(* IEC 61131-3 sources: elnaProjects/ElpcLogic/PomarKc7Changed/build_USO_ecl/_ (part 5) *)

FUNCTION_BLOCK fb_vibegPNSAlg
  VAR_IN_OUT
    StrAlg : struct_Alg;
  END_VAR
  VAR
    autoPnsOff : struct_PhaseAlgoritm;
    waitVibeg : struct_PhaseAlgoritm;
    pnsOff : struct_PhaseAlgoritm;
    vibegEnd : struct_PhaseAlgoritm;
  END_VAR
  VAR_IN_OUT
    algContinue : struct_Question;
  END_VAR
  VAR
    fb_autoPnsOff : fb_ph_algoritm;
    fb_waitVibeg : fb_ph_Timer;
    fb_algContinue : fb_Question;
    fb_pnsOff : fb_ph_Switch;
    fb_vibegEnd : fb_ph_CustomPhase;
    _sunpackerCommand : fb_sunpackerCommand;
    _statusAi : TYPE_StatusAi;
    _Answers : TYPE_Answers;
    _statusDualInput : TYPE_statusDualInput;
    _DualStateImAction : TYPE_DualStateImAction;
    _PhaseAlgoritmAction : TYPE_PhaseAlgoritmAction;
    source : BYTE;
    cmd : BYTE;
    lastCmd : BYTE;
    source_for_Status : BYTE;
    cmd_for_Status : BYTE;
    command_error_for_Status : BYTE;
    resetCmdTimer : TON;
    resetCmdTimerPriznak : BOOL;
    onInit : BOOL;
    waitReset : TON;
  END_VAR
  VAR_EXTERNAL
    IM : ImConfig;
    algoritms : AlgoritmsConfig;
    ai : AiConfig;
    protections : ProtectionsConfig;
    AlgTimers : struct_AlgTimers;
  END_VAR

  IF NOT onInit THEN
   fb_autoPnsOff(phaseNumber:=0, act:=_reset, waitCompletion:=FALSE);
    fb_waitVibeg(phaseNumber:=1, delay:=T#300S);
       algContinue.AnswerVariants:=_Answers.ANS_YES;
       fb_pnsOff(phaseNumber:=2, act:=_off);
     fb_vibegEnd(phaseNumber:=14);
  onInit:=TRUE;
  END_IF;

   fb_autoPnsOff(StrPh:=autoPnsOff, alg:=algoritms.autoPns);
    fb_waitVibeg(StrPh:=waitVibeg, timer:=AlgTimers.vibegPNS_Timer);
  fb_algContinue(StrQ:=algContinue);
       fb_pnsOff(StrPh:=pnsOff, Im:=IM.pns);
     fb_vibegEnd(StrPh:=vibegEnd);

  IF StrAlg.isRuning THEN

  StrAlg.hasError := autoPnsOff.error OR pnsOff.error;

      IF IM.pns.onStatus = _statusDualInput.STATUS_ON AND NOT vibegEnd.top THEN

  	runPhase(vibegEnd);
            runPhase(waitVibeg);
            askQuestion(algContinue);

      END_IF;

      IF waitVibeg.top OR (algContinue.answer = _Answers.ANS_YES) THEN
  	vibegEnd.top:=TRUE;
  	resetPhase(waitVibeg);
            resetQuestion(algContinue);

            resetAiProtection(protections.Os_sdvig_nagnetatelja_minus);
            (*resetDiProtection(protections.Vibro_skorost_OP_shesterni_RED_T6);*)

  	(*IM.SingleSignals.P_oil_low.Disabled_Sig:=TRUE;*)
  	ai.Pmasla_posle_GNS.Disabled_LA:=TRUE;
            ai.Pmasla_posle_GNS.Disabled_LW:=TRUE;
            ai.Pmasla_posle_NU.Disabled_LW:=TRUE;
  	runPhase(pnsOff);
      END_IF;

      StrAlg.isEnded:=pnsOff.top;

  END_IF;

  StrAlg.CanRun := StrAlg.inCanRun;
  StrAlg.OpcCommandsDisabled := StrAlg.inOpcCommandsDisabled;

  (* ---- Если управление с ВУ заблокировано, то  передаем команду из алгоритма ---- *)
  IF StrAlg.inOpcCommandsDisabled THEN
  	StrAlg.inCommand := StrAlg.inCommand_Alg;
  ELSE (* иначе передаем команду с АРМа*)
  	StrAlg.inCommand := StrAlg.inCommand_ARM;
  END_IF;

  _sunpackerCommand(command := StrAlg.inCommand);
  	source := _sunpackerCommand.source;
  	cmd := _sunpackerCommand.cmd;

  IF cmd <> 0 AND lastCmd <> cmd AND (((NOT StrAlg.opcCommandsDisabled) AND source > 0) OR source = 0) then
  	CASE BYTE_TO_INT(cmd) OF
  		(*cmdRun*) 1: 	IF (StrAlg.CanRun) THEN
  					StrAlg.isRuning := TRUE;
  					StrAlg.isEnded := FALSE;
  					StrAlg.hasError := FALSE;
  					(*****************       OnRun       *****************)
                                                    runPhase(autoPnsOff);

  					cmd_for_Status := cmd;
  					source_for_Status := source;
  					command_error_for_Status := 0;
  				ELSE
  					StrAlg.isRuning := FALSE;
  					StrAlg.isEnded := FALSE;
  					StrAlg.hasError 	:= FALSE;

  					cmd_for_Status := 0;
  					source_for_Status := source;
  					command_error_for_Status := cmd;
  				END_IF;
  		(*cmdReset*) 2: 	StrAlg.isRuning := FALSE;
  				StrAlg.isEnded := FALSE;
  				StrAlg.hasError 	:= FALSE;

                                           (*****************       OnReset       *****************)
                                         waitReset(IN:=FALSE);
                                         resetPhase(autoPnsOff);
                                         resetPhase(waitVibeg);
                                         resetPhase(vibegEnd);
                                         resetPhase(pnsOff);
                                         resetQuestion(algContinue);

  				cmd_for_Status := cmd;
  				source_for_Status := source;
  				command_error_for_Status := 0;
  	END_CASE;
  	resetCmdTimer(IN := false);
  	resetCmdTimerPriznak := TRUE;
  END_IF;
  lastCmd := cmd;

  resetCmdTimer(IN := resetCmdTimerPriznak, PT := T#5S);
  IF resetCmdTimer.Q THEN
  	resetCmdTimerPriznak := FALSE;
  	source_for_Status := 0;
  	cmd_for_Status := 0;
  	command_error_for_Status := 0;
  END_IF;

  StrAlg.Start:= autoPnsOff.startStatus
              OR waitVibeg.startStatus
              OR pnsOff.startStatus
              OR vibegEnd.startStatus;

  StrAlg.Error:= autoPnsOff.errorStatus
              OR waitVibeg.errorStatus
              OR pnsOff.errorStatus
              OR vibegEnd.errorStatus;

  StrAlg.Top:=   autoPnsOff.topStatus
              OR waitVibeg.topStatus
              OR pnsOff.topStatus
              OR vibegEnd.topStatus;

  (*TODO: TYPE PROGRAM CODE HERE*)
  StrAlg.status :=  SHL(BYTE_TO_DWORD(source_for_Status), 29)
  			OR SHL(BYTE_TO_DWORD(cmd_for_Status), 26)
  			OR SHL(BYTE_TO_DWORD(command_error_for_Status), 23)
  			OR SHL(BOOL_TO_DWORD(StrAlg.OpcCommandsDisabled ), 21)
  			OR SHL(BOOL_TO_DWORD(StrAlg.hasError),4)
  			OR SHL(BOOL_TO_DWORD(StrAlg.CanRun),2)
  			OR SHL(BOOL_TO_DWORD(StrAlg.isEnded),1)
  			OR BOOL_TO_DWORD(StrAlg.isRuning);
END_FUNCTION_BLOCK

FUNCTION_BLOCK fb_AutoNUAlg
  VAR_IN_OUT
    StrAlg : struct_Alg;
    nu1 : struct_OilPump;
    nu2 : struct_OilPump;
  END_VAR
  VAR_INPUT
    dPoil : struct_AI;
  END_VAR
  VAR_IN_OUT
    mainNU : struct_DiscretParametr;
    Lowdp_di : struct_singleSignal;
    Ust_Swap : struct_AnalogParametr;
  END_VAR
  VAR
    _prevMainNU : UINT;
    _sunpackerCommand : fb_sunpackerCommand;
    _statusAi : TYPE_StatusAi;
    _statusDualInput : TYPE_statusDualInput;
    _commandDualInput : TYPE_commandDualInput;
    source : BYTE;
    cmd : BYTE;
    lastCmd : BYTE;
    source_for_Status : BYTE;
    cmd_for_Status : BYTE;
    command_error_for_Status : BYTE;
    resetCmdTimer : TON;
    waitPressure : TON;
    waitPressureTrig : R_TRIG;
    resetCmdTimerPriznak : BOOL;
    onInit : BOOL;
    onStart : BOOL;
  END_VAR
  VAR_EXTERNAL
    NotHasRezervNU : BOOL;
    Reset_HasNU : BOOL;
  END_VAR

  IF NOT onInit THEN
  StrAlg.inCanRun:=TRUE;
  StrAlg.inOpcCommandsDisabled:=TRUE;
  (*nu1.Osnovnoy:=TRUE; nu2.Osnovnoy:=FALSE;*)
  onInit:=TRUE;
  END_IF;

  IF Reset_HasNU THEN
  nu1.inBlocked:=FALSE;
  nu2.inBlocked:=FALSE;
  END_IF;

  NotHasRezervNU:=(nu1.Blocked OR nu2.Blocked);

  IF StrAlg.isRuning THEN

  StrAlg.hasError := nu1.CommandFault OR nu2.CommandFault OR (dPoil.interval<_statusAi.normal);

   IF mainNU.value<>_prevMainNU OR NOT onStart THEN

          CASE mainNU.value OF
  	0: nu1.Osnovnoy:=TRUE; nu2.Osnovnoy:=FALSE;
  	1: nu1.Osnovnoy:=FALSE; nu2.Osnovnoy:=TRUE;

          END_CASE;

      IF  nu1.Osnovnoy AND NOT nu1.Blocked THEN
          nu1.inCommand_Alg:=BYTE_TO_WORD(_commandDualInput.CMD_ON);
      ELSIF NOT NotHasRezervNU THEN
          nu1.inCommand_Alg:=BYTE_TO_WORD(_commandDualInput.CMD_OFF);
      END_IF;

      IF  nu2.Osnovnoy AND NOT nu2.Blocked THEN
          nu2.inCommand_Alg:=BYTE_TO_WORD(_commandDualInput.CMD_ON);
       ELSIF NOT NotHasRezervNU THEN
          nu2.inCommand_Alg:=BYTE_TO_WORD(_commandDualInput.CMD_OFF);
      END_IF;
        onStart:=TRUE;
       _prevMainNU:=mainNU.value;
   END_IF;

    (*IF (nu1.onStatus = _statusDualInput.STATUS_On) OR (nu2.onStatus = _statusDualInput.STATUS_On) THEN*)
      (*Если через 5С насос не нагнал 100кПа масла - он сломался и надо переключить насос*)
      IF dPoil.interval>= _statusAi.NORMAL THEN
            waitPressure(IN:=(dPoil.value<Ust_Swap.Value OR LowdP_DI.q) AND NOT NotHasRezervNU, PT:= T#5S);
      ELSE
  	waitPressure(IN:=(FALSE));
      END_IF;

      waitPressureTrig(CLK:=waitPressure.Q);
      IF waitPressureTrig.Q THEN
  	(*IF nu1.onStatus = _statusDualInput.STATUS_ON THEN*)
             IF mainNU.value = 0 THEN
  		nu1.inBlocked:=TRUE;
                      nu1.inCommand_Alg:=BYTE_TO_WORD(_commandDualInput.CMD_OFF);
  			(*IF 	mainNU.value = 0 THEN*)
                                          setValue(mainNU, 1);
  			(*END_IF;*)
  	END_IF;

  	(*IF nu2.onStatus = _statusDualInput.STATUS_ON THEN*)
            IF mainNU.value = 1 THEN
  		nu2.inBlocked:=TRUE;
                      nu2.inCommand_Alg:=BYTE_TO_WORD(_commandDualInput.CMD_OFF);
  			(*IF 	mainNU.value = 1 THEN*)
  				setValue(mainNU, 0);
  			(*END_IF;*)
  	END_IF;
      END_IF;
   (* END_IF;*)

  END_IF;

  StrAlg.CanRun := StrAlg.inCanRun;

  StrAlg.OpcCommandsDisabled := StrAlg.inOpcCommandsDisabled;

  (* ---- Если управление с ВУ заблокировано, то  передаем команду из алгоритма ---- *)
  IF StrAlg.inOpcCommandsDisabled THEN
  	StrAlg.inCommand := StrAlg.inCommand_Alg;
  ELSE (* иначе передаем команду с АРМа*)
  	StrAlg.inCommand := StrAlg.inCommand_ARM;
  END_IF;

  _sunpackerCommand(command := StrAlg.inCommand);
  	source := _sunpackerCommand.source;
  	cmd := _sunpackerCommand.cmd;

  IF cmd <> 0 AND lastCmd <> cmd AND (((NOT StrAlg.opcCommandsDisabled) AND source > 0) OR source = 0) then
  	CASE BYTE_TO_INT(cmd) OF
  		(*cmdRun*) 1: 	IF (StrAlg.CanRun) THEN
  					StrAlg.isRuning := TRUE;
  					StrAlg.isEnded := FALSE;
  					StrAlg.hasError := FALSE;

                                                    (*****************       OnRun       *****************)
  					nu1.inOpcCommandsDisabled:=TRUE;
                                                    nu2.inOpcCommandsDisabled:=TRUE;

  					cmd_for_Status := cmd;
  					source_for_Status := source;
  					command_error_for_Status := 0;
  				ELSE
  					StrAlg.isRuning := FALSE;
  					StrAlg.isEnded := FALSE;
  					StrAlg.hasError 	:= FALSE;

  					cmd_for_Status := 0;
  					source_for_Status := source;
  					command_error_for_Status := cmd;
  				END_IF;
  		(*cmdReset*) 2: 	StrAlg.isRuning := FALSE;
  				StrAlg.isEnded := FALSE;
  				StrAlg.hasError 	:= FALSE;

                                          (*****************       OnReset       *****************)
                                          waitPressure(IN:=(FALSE));
                                          onStart:=FALSE;

  				cmd_for_Status := cmd;
  				source_for_Status := source;
  				command_error_for_Status := 0;
  	END_CASE;
  	resetCmdTimer(IN := false);
  	resetCmdTimerPriznak := TRUE;
  END_IF;
  lastCmd := cmd;

  resetCmdTimer(IN := resetCmdTimerPriznak, PT := T#5S);
  IF resetCmdTimer.Q THEN
  	resetCmdTimerPriznak := FALSE;
  	source_for_Status := 0;
  	cmd_for_Status := 0;
  	command_error_for_Status := 0;
  END_IF;

  (*TODO: TYPE PROGRAM CODE HERE*)
  StrAlg.status :=  SHL(BYTE_TO_DWORD(source_for_Status), 29)
  			OR SHL(BYTE_TO_DWORD(cmd_for_Status), 26)
  			OR SHL(BYTE_TO_DWORD(command_error_for_Status), 23)
  			OR SHL(BOOL_TO_DWORD(StrAlg.OpcCommandsDisabled ), 21)
                                OR SHL(BOOL_TO_DWORD(NotHasRezervNU), 15)
  			OR SHL(BOOL_TO_DWORD(StrAlg.hasError),4)
  			OR SHL(BOOL_TO_DWORD(StrAlg.CanRun),2)
  			OR SHL(BOOL_TO_DWORD(StrAlg.isEnded),1)
  			OR BOOL_TO_DWORD(StrAlg.isRuning);
END_FUNCTION_BLOCK

FUNCTION_BLOCK fb_ph_WaitAnalogValue
  VAR_IN_OUT
    ai : struct_AI;
  END_VAR
  VAR_INPUT
    more : LREAL;
    less : LREAL;
    PhaseNumber : UINT;
  END_VAR
  VAR_IN_OUT
    StrPh : struct_PhaseAlgoritm;
  END_VAR
  VAR
    CommandFault_Trig : R_TRIG;
    reset_Trig : R_TRIG;
    _statusAi : TYPE_StatusAi;
    _statusDualInput : TYPE_statusDualInput;
  END_VAR

  IF StrPh.run AND NOT StrPh.start THEN
  	StrPh.start := TRUE;
  	StrPh.top := FALSE;
  	StrPh.error := FALSE;
            StrPh.run:=FALSE;
  END_IF;

  IF StrPh.start AND NOT StrPh.top THEN
                      IF ai.interval < _statusAi.normal THEN
  	              StrPh.error := TRUE;
                          StrPh.top:=FALSE;
                      ELSE
                              IF (more<>0.0) OR (less<>0.0) THEN
                              StrPh.top:=TRUE;
  	                    IF more<>0.0 THEN StrPh.top:=StrPh.top AND (ai.value > more); END_IF;
  	                    IF less<>0.0 THEN StrPh.top:=StrPh.top AND (ai.value < less); END_IF;
                              ELSE
  	                  StrPh.top:=TRUE;
                              END_IF;
                     END_IF;
  END_IF;

  IF StrPh.top THEN
  StrPh.error := FALSE;
  END_IF;

  reset_Trig(CLK := StrPh.reset);
  IF reset_Trig.Q THEN
  	StrPh.start := FALSE;
  	StrPh.error := FALSE;
  	StrPh.top := FALSE;
            StrPh.run:=FALSE;
            StrPh.reset:=FALSE;
  END_IF;

  StrPh.startStatus := SHL(BOOL_TO_DWORD(StrPh.start), PhaseNumber);
  StrPh.errorStatus := SHL(BOOL_TO_DWORD(StrPh.error), PhaseNumber);
  StrPh.topStatus := SHL(BOOL_TO_DWORD(StrPh.top), PhaseNumber);
END_FUNCTION_BLOCK

FUNCTION resetAndDisable : BOOL
  VAR_IN_OUT
    alg : struct_Alg;
  END_VAR
  VAR CONSTANT
    cmdReset : WORD      := 2;
  END_VAR

  IF alg.isRuning THEN
                      alg.inOpcCommandsDisabled:=TRUE;
  		alg.inCommand_Alg:=cmdReset;
  END_IF;

   alg.inCanRun:=FALSE;
END_FUNCTION

FUNCTION_BLOCK fb_puskOilSystemAlg
  VAR_IN_OUT
    StrAlg : struct_Alg;
  END_VAR
  VAR
    pnsOn : struct_PhaseAlgoritm;
    LowOil : struct_PhaseAlgoritm;
    BreakPuskTimer_Poil : struct_PhaseAlgoritm;
    Poil_DefenseActive : struct_PhaseAlgoritm;
    autoNuOn : struct_PhaseAlgoritm;
    nuOn : struct_PhaseAlgoritm;
    nu1On : struct_PhaseAlgoritm;
    nu2On : struct_PhaseAlgoritm;
    di_dPmg : struct_PhaseAlgoritm;
    dP_oilGas100 : struct_PhaseAlgoritm;
    runProtect_dP : struct_PhaseAlgoritm;
    testUnsuccessful : struct_PhaseAlgoritm;
    fb_pnsOn : fb_ph_Switch;
    fb_LowOil : fb_ph_WaitAnalogValue;
    fb_BreakPuskTimer_Poil : fb_ph_Timer;
    fb_Poil_DefenseActive : fb_ph_CustomPhase;
    fb_nuOn : fb_ph_CustomPhase;
    fb_nu1On : fb_ph_OilPump;
    fb_nu2On : fb_ph_OilPump;
    fb_autoNuOn : fb_ph_algoritm;
    fb_di_dPmg : fb_ph_CustomPhase;
    fb_dP_oilGas100 : fb_ph_WaitAnalogValue;
    fb_runProtect_dP : fb_ph_CustomPhase;
    fb_testUnsuccessful : fb_ph_CustomPhase;
    _sunpackerCommand : fb_sunpackerCommand;
    _statusAi : TYPE_StatusAi;
    _Answers : TYPE_Answers;
    _statusDualInput : TYPE_statusDualInput;
    _DualStateImAction : TYPE_DualStateImAction;
    _PhaseAlgoritmAction : TYPE_PhaseAlgoritmAction;
    source : BYTE;
    cmd : BYTE;
    lastCmd : BYTE;
    source_for_Status : BYTE;
    cmd_for_Status : BYTE;
    command_error_for_Status : BYTE;
    resetCmdTimer : TON;
    resetCmdTimerPriznak : BOOL;
    onInit : BOOL;
    waitReset : TON;
  END_VAR
  VAR_EXTERNAL
    IM : ImConfig;
    algoritms : AlgoritmsConfig;
    ai : AiConfig;
    protections : ProtectionsConfig;
    AlgTimers : struct_AlgTimers;
  END_VAR

  IF NOT onInit THEN
                 fb_pnsOn(phaseNumber:=0, act:=_on);
                fb_LowOil(phaseNumber:=1);
   fb_BreakPuskTimer_Poil(phaseNumber:=3, delay:=T#240S);
    fb_Poil_DefenseActive(phaseNumber:=5);
                  fb_nuOn(phaseNumber:=6);
                 fb_nu1On(phaseNumber:=11, act:=_on);
                 fb_nu2On(phaseNumber:=12, act:=_on);
              fb_autoNuOn(phaseNumber:=7, act:=_run, waitCompletion:=FALSE);
               fb_di_dPmg(phaseNumber:=8);
          fb_dP_oilGas100(phaseNumber:=9);
         fb_runProtect_dP(phaseNumber:=10);
      fb_testUnsuccessful(phaseNumber:=17);

  onInit:=TRUE;
  END_IF;

                fb_pnsOn(StrPh:=pnsOn, Im:=IM.pns);
               (*fb_LowOil(StrPh:=LowOil, ai:=ai.Pmasla_posle_GNS, more:=im.AutoPns_UstRun.Value);*)
  fb_BreakPuskTimer_Poil(StrPh:=BreakPuskTimer_Poil, timer:=AlgTimers.puskOilSystem_BreakPuskTimer_Poil);
   fb_Poil_DefenseActive(StrPh:=Poil_DefenseActive);
                 fb_nuOn(StrPh:=nuOn);
                fb_nu1On(StrPh:=nu1On, Im:=Im.nu1);
                fb_nu2On(StrPh:=nu2On, Im:=Im.nu2);
             fb_autoNuOn(StrPh:=autoNuOn, alg:=algoritms.autoNu);
              fb_di_dPmg(StrPh:=di_dPmg);
         (*fb_dP_oilGas100(StrPh:=dP_oilGas100, ai:=ai.Tmasla_MB, more:=im.PuskOilSystem_UstdPmg.Value);*)
        fb_runProtect_dP(StrPh:=runProtect_dP);
     fb_testUnsuccessful(StrPh:=testUnsuccessful);

  IF StrAlg.isRuning THEN

      StrAlg.hasError := LowOil.error OR dP_oilGas100.error OR pnsOn.error OR testUnsuccessful.error;

      IF pnsOn.top THEN
          runPhase(LowOil);
      END_IF;

      IF LowOil.top THEN
          runAiProtection(protections.Os_sdvig_nagnetatelja_minus);
          (*runDiProtection(protections.Vibro_skorost_OP_shesterni_RED_T6);*)
          runPhase(Poil_DefenseActive);
          (*IM.SingleSignals.P_oil_low.Disabled_Sig:=FALSE;*)
          ai.Pmasla_posle_GNS.Disabled_LA:=FALSE;
          ai.Pmasla_posle_GNS.Disabled_LW:=FALSE;
          ai.Pmasla_posle_NU.Disabled_LW:=FALSE;
      END_IF;

      IF Poil_DefenseActive.start AND NOT Poil_DefenseActive.top THEN
         Poil_DefenseActive.top:=protections.Os_sdvig_nagnetatelja_minus.isRunning AND protections.Vibro_skorost_OP_shesterni_RED_T6.isRunning;
      END_IF;

      IF Poil_DefenseActive.top THEN
         (* runPhase(autoNuOn);*)
  	runPhase(nuOn);
      END_IF;

      IF nuOn.start AND NOT nuOn.top THEN
         (* IF IM.SingleOutputs.Value = 0 THEN
              runPhase(nu1On);
          END_IF;

          IF IM.SingleOutputs.Value = 1 THEN
              runPhase(nu2On);
          END_IF;*)
         nuOn.top:= Im.nu1.onStatus = _statusDualInput.STATUS_ON OR Im.nu2.onStatus = _statusDualInput.STATUS_ON;
      END_IF;

      IF nuOn.top THEN
  	runPhase(di_dPmg);
            runPhase(dP_oilGas100);
      END_IF;

      (*IF di_dPmg.start AND NOT di_dPmg.top THEN
         di_dPmg.top:= NOT IM.SingleSignals.dP_oilgaz_low.Q;
      END_IF;*)

      IF dP_oilGas100.top AND di_dPmg.top THEN
            runPhase(autoNuOn);
  	runPhase(runProtect_dP);
  	runAiProtection(protections.Os_sdvig_nagnetatelja_plus);
            (*runDiProtection(protections.Vibro_skorost_OP_shesterni_RED_T5);
            IM.SingleSignals.dP_oilgaz_low.Disabled_Sig:=FALSE;
            ai.Tmasla_MB.Disabled_LA:=FALSE;
            ai.Tmasla_MB.Disabled_LW:=FALSE;*)
      END_IF;

      IF runProtect_dP.start AND NOT runProtect_dP.top THEN
         runProtect_dP.top:= protections.Os_sdvig_nagnetatelja_plus.isRunning AND protections.Vibro_skorost_OP_shesterni_RED_T5.isRunning;
      END_IF;

      IF BreakPuskTimer_Poil.top AND (NOT runProtect_dP.top) THEN
  	testUnsuccessful.error:=TRUE;
      END_IF;

      IF runProtect_dP.top THEN
            resetPhase(BreakPuskTimer_Poil);
  	waitReset(IN:=TRUE);
      END_IF;

      IF waitReset.Q AND NOT (algoritms.Apusk.isRuning OR algoritms.SemiAutoPusk.isRuning) THEN
      resetAndDisable(StrAlg);
      END_IF;

      StrAlg.isEnded:=runProtect_dP.top;
  END_IF;

  StrAlg.CanRun := StrAlg.inCanRun;
  StrAlg.OpcCommandsDisabled := StrAlg.inOpcCommandsDisabled;

  (* ---- Если управление с ВУ заблокировано, то  передаем команду из алгоритма ---- *)
  IF StrAlg.inOpcCommandsDisabled THEN
  	StrAlg.inCommand := StrAlg.inCommand_Alg;
  ELSE (* иначе передаем команду с АРМа*)
  	StrAlg.inCommand := StrAlg.inCommand_ARM;
  END_IF;

  _sunpackerCommand(command := StrAlg.inCommand);
  	source := _sunpackerCommand.source;
  	cmd := _sunpackerCommand.cmd;

  IF cmd <> 0 AND lastCmd <> cmd AND (((NOT StrAlg.opcCommandsDisabled) AND source > 0) OR source = 0) then
  	CASE BYTE_TO_INT(cmd) OF
  		(*cmdRun*) 1: 	IF (StrAlg.CanRun) THEN
  					StrAlg.isRuning := TRUE;
  					StrAlg.isEnded := FALSE;
  					StrAlg.hasError := FALSE;
  					(*****************       OnRun       *****************)
                                                    runPhase(pnsOn);
                                                    runPhase(BreakPuskTimer_Poil);
                                                    runPhase(testUnsuccessful);
  					cmd_for_Status := cmd;
  					source_for_Status := source;
  					command_error_for_Status := 0;
  				ELSE
  					StrAlg.isRuning := FALSE;
  					StrAlg.isEnded := FALSE;
  					StrAlg.hasError 	:= FALSE;

  					cmd_for_Status := 0;
  					source_for_Status := source;
  					command_error_for_Status := cmd;
  				END_IF;
  		(*cmdReset*) 2: 	StrAlg.isRuning := FALSE;
  				StrAlg.isEnded := FALSE;
  				StrAlg.hasError 	:= FALSE;

                                           (*****************       OnReset       *****************)
                                          waitReset(IN:=FALSE);
                                          resetPhase(pnsOn);
                                          resetPhase(LowOil);
                                          resetPhase(BreakPuskTimer_Poil);
                                          resetPhase(Poil_DefenseActive);
                                          resetPhase(autoNuOn);
                                          resetPhase(nu1On);
                                          resetPhase(nu2On);
                                          resetPhase(nuOn);
                                          resetPhase(di_dPmg);
                                          resetPhase(dP_oilGas100);
                                          resetPhase(runProtect_dP);
                                          resetPhase(testUnsuccessful);
  	                              (*protections.Os_sdvig_nagnetatelja_minus.inOpcCommandsDisabled:=FALSE;
                                          protections.Vibro_skorost_OP_shesterni_RED_T6.inOpcCommandsDisabled:=FALSE;
                                          protections.Os_sdvig_nagnetatelja_plus.inOpcCommandsDisabled:=FALSE;
                                          protections.Vibro_skorost_OP_shesterni_RED_T5.inOpcCommandsDisabled:=FALSE;*)

  				cmd_for_Status := cmd;
  				source_for_Status := source;
  				command_error_for_Status := 0;
  	END_CASE;
  	resetCmdTimer(IN := false);
  	resetCmdTimerPriznak := TRUE;
  END_IF;
  lastCmd := cmd;

  resetCmdTimer(IN := resetCmdTimerPriznak, PT := T#5S);
  IF resetCmdTimer.Q THEN
  	resetCmdTimerPriznak := FALSE;
  	source_for_Status := 0;
  	cmd_for_Status := 0;
  	command_error_for_Status := 0;
  END_IF;

  StrAlg.Start:= pnsOn.startStatus
              OR LowOil.startStatus
              OR BreakPuskTimer_Poil.startStatus
              OR Poil_DefenseActive.startStatus
              OR nuOn.startStatus
              OR di_dPmg.startStatus
              OR dP_oilGas100.startStatus
              OR runProtect_dP.startStatus
              OR testUnsuccessful.startStatus;

  StrAlg.Error:= pnsOn.errorStatus
              OR LowOil.errorStatus
              OR BreakPuskTimer_Poil.errorStatus
              OR Poil_DefenseActive.errorStatus
              OR nuOn.errorStatus
              OR di_dPmg.errorStatus
              OR dP_oilGas100.errorStatus
              OR runProtect_dP.errorStatus
              OR testUnsuccessful.errorStatus;

  StrAlg.Top:=   pnsOn.topStatus
              OR LowOil.topStatus
              OR BreakPuskTimer_Poil.topStatus
              OR Poil_DefenseActive.topStatus
              OR nuOn.topStatus
              OR di_dPmg.topStatus
              OR dP_oilGas100.topStatus
              OR runProtect_dP.topStatus
              OR testUnsuccessful.topStatus;

  (*TODO: TYPE PROGRAM CODE HERE*)
  StrAlg.status :=  SHL(BYTE_TO_DWORD(source_for_Status), 29)
  			OR SHL(BYTE_TO_DWORD(cmd_for_Status), 26)
  			OR SHL(BYTE_TO_DWORD(command_error_for_Status), 23)
  			OR SHL(BOOL_TO_DWORD(StrAlg.OpcCommandsDisabled ), 21)
  			OR SHL(BOOL_TO_DWORD(StrAlg.hasError),4)
  			OR SHL(BOOL_TO_DWORD(StrAlg.CanRun),2)
  			OR SHL(BOOL_TO_DWORD(StrAlg.isEnded),1)
  			OR BOOL_TO_DWORD(StrAlg.isRuning);
END_FUNCTION_BLOCK

FUNCTION_BLOCK NOAlg
  VAR_IN_OUT
    StrAlg : struct_Alg;
  END_VAR
  VAR
    timer120 : struct_PhaseAlgoritm;
    kran6Open : struct_PhaseAlgoritm;
    pnsOn : struct_PhaseAlgoritm;
    kran4Close : struct_PhaseAlgoritm;
    kran3bOpen : struct_PhaseAlgoritm;
    mvOff : struct_PhaseAlgoritm;
    kran1Close : struct_PhaseAlgoritm;
    kran2Close : struct_PhaseAlgoritm;
    kran3Close : struct_PhaseAlgoritm;
    kran5Open : struct_PhaseAlgoritm;
    error_Krans : struct_PhaseAlgoritm;
    autoPnsOff : struct_PhaseAlgoritm;
    Pg_VhodLessThen300 : struct_PhaseAlgoritm;
    Pg_VyhodLessThen300 : struct_PhaseAlgoritm;
    nu1off : struct_PhaseAlgoritm;
    nu2off : struct_PhaseAlgoritm;
    AutoNU_Off : struct_PhaseAlgoritm;
    timer600 : struct_PhaseAlgoritm;
    pnsOff : struct_PhaseAlgoritm;
    Avom1Off : struct_PhaseAlgoritm;
    Avom2Off : struct_PhaseAlgoritm;
    Avom3Off : struct_PhaseAlgoritm;
    Avom4Off : struct_PhaseAlgoritm;
    autoAVOMOff : struct_PhaseAlgoritm;
    timer5 : struct_PhaseAlgoritm;
    klapan1 : struct_PhaseAlgoritm;
    klapan2 : struct_PhaseAlgoritm;
    nu_On : struct_PhaseAlgoritm;
    fb_timer120 : fb_ph_Timer;
    fb_kran6Open : fb_ph_Kran;
    fb_pnsOn : fb_ph_Switch;
    fb_kran4Close : fb_ph_Kran;
    fb_kran3bOpen : fb_ph_Kran;
    fb_mvOff : fb_ph_SectionSwitch;
    fb_kran1Close : fb_ph_Kran;
    fb_kran2Close : fb_ph_Kran;
    fb_kran3Close : fb_ph_Kran;
    fb_kran5Open : fb_ph_Kran;
    fb_error_Krans : fb_ph_CustomPhase;
    fb_autoPnsOff : fb_ph_algoritm;
    fb_Pg_VhodLessThen300 : fb_ph_CustomPhase;
    fb_Pg_VyhodLessThen300 : fb_ph_CustomPhase;
    fb_nu1Off : fb_ph_OilPump;
    fb_nu2Off : fb_ph_OilPump;
    fb_autoNuOff : fb_ph_algoritm;
    fb_timer600 : fb_ph_Timer;
    fb_pnsOff : fb_ph_Switch;
    fb_Avom1Off : fb_ph_Switch;
    fb_Avom2Off : fb_ph_Switch;
    fb_Avom3Off : fb_ph_Switch;
    fb_Avom4Off : fb_ph_Switch;
    fb_autoAVOMOff : fb_ph_algoritm;
    fb_timer5 : fb_ph_Timer;
    fb_klapan1 : fb_ph_CustomPhase;
    fb_klapan2 : fb_ph_CustomPhase;
    fb_nu_On : fb_ph_CustomPhase;
    _sunpackerCommand : fb_sunpackerCommand;
    _statusAi : TYPE_StatusAi;
    _Answers : TYPE_Answers;
    _statusDualInput : TYPE_statusDualInput;
    _commandDualInput : TYPE_commandDualInput;
    _DualStateImAction : TYPE_DualStateImAction;
    _PhaseAlgoritmAction : TYPE_PhaseAlgoritmAction;
    source : BYTE;
    cmd : BYTE;
    lastCmd : BYTE;
    source_for_Status : BYTE;
    cmd_for_Status : BYTE;
    command_error_for_Status : BYTE;
    resetCmdTimer : TON;
    resetCmdTimerPriznak : BOOL;
    onInit : BOOL;
    waitReset : TON;
  END_VAR
  VAR_EXTERNAL
    IM : ImConfig;
    algoritms : AlgoritmsConfig;
    ai : AiConfig;
    protections : ProtectionsConfig;
    ModeGpa : TYPE_ModeGpa;
    algManager : struct_AlgoritmsManager;
    AlgTimers : struct_AlgTimers;
  END_VAR
  VAR CONSTANT
    Ust_Pgaza : LREAL      := 0.3;
  END_VAR

  IF NOT onInit THEN
      fb_timer120(phaseNumber:=1, delay:=T#120S);
      fb_kran6Open(phaseNumber:=2, act:=_on);
      fb_kran4Close(phaseNumber:=3, act:=_off);
      fb_kran3bOpen(phaseNumber:=4, act:=_off);
      fb_mvOff(phaseNumber:=5, act:=_off);
      fb_kran1Close(phaseNumber:=6, act:=_off);
      fb_kran2Close(phaseNumber:=7, act:=_off);
      fb_kran3Close(phaseNumber:=8, act:=_off);
      fb_kran5Open(phaseNumber:=9, act:=_on);
      fb_error_Krans(phaseNumber:=10);
      fb_autoPnsOff(phaseNumber:=11, act:=_reset, waitCompletion:=FALSE);
      fb_pnsOn(phaseNumber:=12, act:=_on);
      fb_Pg_VhodLessThen300(phaseNumber:=13);
      fb_Pg_VyhodLessThen300(phaseNumber:=14);
      fb_nu1Off(phaseNumber:=15, act:=_off);
      fb_nu2Off(phaseNumber:=16, act:=_off);
      fb_autoNuOff(phaseNumber:=17, act:=_reset, waitCompletion:=FALSE);
      fb_timer600(phaseNumber:=18, delay:=T#600S);
      fb_pnsOff(phaseNumber:=19, act:=_off);
      fb_Avom1Off(phaseNumber:=20, act:=_off);
      fb_Avom2Off(phaseNumber:=21, act:=_off);
      fb_Avom3Off(phaseNumber:=22, act:=_off);
      fb_Avom4Off(phaseNumber:=23, act:=_off);
      fb_autoAVOMOff(phaseNumber:=24, act:=_reset, waitCompletion:=FALSE);
      fb_timer5(phaseNumber:=25, delay:=T#5S);
      fb_klapan1(phaseNumber:=26);
      fb_klapan2(phaseNumber:=27);
      fb_nu_On(phaseNumber:=28);

  onInit:=TRUE;
  END_IF;

  fb_timer120(StrPh:=timer120, timer:=AlgTimers.No_wait120);
  fb_kran6Open(StrPh:=kran6Open, Im:=Im.kran6);
  fb_pnsOn(StrPh:=pnsOn, Im:=Im.pns);
  fb_kran4Close(StrPh:=kran4Close, Im:=Im.kran4);
  fb_kran3bOpen(StrPh:=kran3bOpen, Im:=Im.kran3b);
  fb_mvOff(StrPh:=mvOff, Im:=Im.mv);
  fb_kran1Close(StrPh:=kran1Close, Im:=Im.kran1);
  fb_kran2Close(StrPh:=kran2Close, Im:=Im.Kran2);
  fb_kran3Close(StrPh:=kran3Close, Im:=Im.Kran3);
  fb_kran5Open(StrPh:=kran5Open, Im:=Im.Kran5);
  fb_error_Krans(StrPh:=error_Krans);
  fb_autoPnsOff(StrPh:=autoPnsOff, alg:=algoritms.autoPns);
  fb_Pg_VhodLessThen300(StrPh:=Pg_VhodLessThen300);
  fb_Pg_VyhodLessThen300(StrPh:=Pg_VyhodLessThen300);
  fb_nu1Off(StrPh:=nu1off, Im:=Im.nu1);
  fb_nu2Off(StrPh:=nu2off, Im:=Im.nu2);
  fb_autoNuOff(StrPh:=AutoNU_Off, alg:=algoritms.autoNu);
  fb_timer600(StrPh:=timer600, timer:=AlgTimers.No_wait600);
  fb_pnsOff(StrPh:=pnsOff, Im:=Im.pns);
  fb_Avom1Off(StrPh:=Avom1Off, Im:=Im.v1_Avom);
  fb_Avom2Off(StrPh:=Avom2Off, Im:=Im.v2_Avom);
  fb_Avom3Off(StrPh:=Avom3Off, Im:=Im.v3_Avom);
  fb_Avom4Off(StrPh:=Avom4Off, Im:=Im.v4_Avom);
  fb_autoAVOMOff(StrPh:=autoAVOMOff, alg:=algoritms.AutoAvom);
  fb_timer5(StrPh:=timer5, timer:=AlgTimers.No_wait5);
  fb_klapan1(StrPh:=klapan1);
  fb_klapan2(StrPh:=klapan2);
  fb_nu_On(StrPh:=nu_On);

  StrAlg.CanRun := StrAlg.inCanRun;
  StrAlg.OpcCommandsDisabled := StrAlg.inOpcCommandsDisabled;

  IF StrAlg.isRuning THEN
      (* кран 6 не открыт - запуск таймера *)
      IF NOT kran6Open.top AND NOT timer120.top  THEN
  	runPhase(timer120);
      ELSE
      (* счетчик отработал и кран 6 не открыт - ошибка *)
          IF timer120.top AND NOT kran6Open.top THEN
              error_Krans.error := TRUE;
          END_IF;
      END_IF;

      (* старт смазки кранов *)
      IF (*algoritms.F3.Smazka_1_2 OR *)IM.kran1.onStatus = _statusDualInput.STATUS_ON OR IM.kran1.onStatus = _statusDualInput.STATUS_TRANSITIONAL
  	OR IM.kran2.onStatus = _statusDualInput.STATUS_ON OR IM.kran2.onStatus = _statusDualInput.STATUS_TRANSITIONAL  THEN
          IF (*(algoritms.F3.Smazka_1_2 OR *)IM.kran1.onStatus = _statusDualInput.STATUS_ON OR IM.kran1.onStatus = _statusDualInput.STATUS_TRANSITIONAL AND NOT klapan1.start AND NOT kran1Close.top THEN
              runPhase(klapan1);
          END_IF;
          IF (*(algoritms.F3.Smazka_1_2 OR *)IM.kran2.onStatus = _statusDualInput.STATUS_ON OR IM.kran2.onStatus = _statusDualInput.STATUS_TRANSITIONAL AND NOT klapan2.start AND NOT kran2Close.top THEN
              runPhase(klapan2);
          END_IF;
      (*algoritms.F3.Smazka_1_2:=FALSE;*)
      END_IF;

      (* открыть кран 6 кран 4 *)
      runPhase(kran6Open);
      runPhase(kran4Close);

      (*не понимаю
      IF kran4Close.top THEN
          ystavki.Block_kr4_alg.setValue (0);
      END_IF;*)

      (* кран 6 открыт *)
      IF kran6Open.top THEN
  	runPhase(kran3bOpen);
  	resetPhase(timer120);
  	(*error_Krans.top := FALSE;
  	error_Krans.error := FALSE;*)
  	(*algoritms.S_Vibr.CanRun:=FALSE;
  	algoritms.S_Vibr.reset (); net takogo alg*)
      END_IF;
      IF kran3bOpen.top AND NOT mvoff.start THEN
  	resetDiProtection(protections.mvOff);
  	resetDiProtection(protections.Off_avar_vikluchatel);
  	resetDiProtection(protections.Reg_vozb_off);
  	runPhase(mvOff);
      END_IF;

      IF mvOff.top (*AND NOT flag1*) THEN
          algoritms.AutoPns.inCanRun :=FALSE;
          (*algoritms.AutoPNS_Start.reset (); nichego ne ponimau
          algoritms.AutoPns.inCanRun :=FALSE;*)
          runPhase(autoPnsOff);
          runPhase(pnsOn);
          resetDiProtection(protections.Kran1_sdvig);
          resetDiProtection(protections.Kran2_sdvig);
          runPhase(kran1Close);
          runPhase(kran2Close);
          runPhase(kran3Close);
          runPhase(nu_On);

          (*тут запустить насосы уплотнения *)

          (*algoritms.autoNu.inCanRun:=FALSE;
          algoritms.autoNu_2.reset ();
          algoritms.autoNu_1.inCanRun:=TRUE;
          algoritms.autoNu_1.run ();
          flag1:=TRUE; что тут происходит?*)
      END_IF;
      IF ((IM.nu1.onStatus =_statusDualInput.STATUS_ON) OR (IM.nu2.onStatus =_statusDualInput.STATUS_ON)) AND nu_On.start AND NOT nu_On.top THEN
          nu_On.top:=TRUE;
      END_IF;

      (* выдача смазки *)
      IF klapan1.start AND kran1Close.top THEN
          (*IM.Kr1_Smazka.impulse(); не понимаю((((((((*)
          klapan1.top:=TRUE;
      END_IF;

      IF klapan2.start AND kran2Close.top THEN
  	(*IM.Kr2_Smazka.impulse(); не понимаю *)
  	klapan2.top:=TRUE;
      END_IF;

      (* кран 1 кран 2 кран 3 кран 4 закрыты - открыть кран 5 *)
      IF kran1Close.top AND kran2Close.top AND kran3Close.top AND kran4Close.top THEN
          runPhase(kran5Open);
          resetAiProtection(protections.Pgaza_na_vyhode_nagnetatelia);
      END_IF;

      IF kran5Open.top THEN
          runPhase(Pg_VhodLessThen300);
          runPhase(Pg_VyhodLessThen300);
      END_IF;

      IF Pg_VhodLessThen300.start AND NOT Pg_VhodLessThen300.top THEN
          IF (ai.Pgaza_na_vhode_nagnetatelia.interval>= _statusAi.NORMAL) AND (ai.Pgaza_na_vhode_nagnetatelia.value < 0.3) THEN
              Pg_VhodLessThen300.top:=TRUE;
          END_IF;
      END_IF;

      IF Pg_VyhodLessThen300.start AND NOT Pg_VyhodLessThen300.top THEN
          IF (ai.Pgaza_na_vyhode_nagnetatelia.interval>=_statusAi.NORMAL) AND (ai.Pgaza_na_vyhode_nagnetatelia.value < 0.3) THEN
              Pg_VyhodLessThen300.top:=TRUE;
          END_IF;
      END_IF;

      IF Pg_VhodLessThen300.top AND Pg_VyhodLessThen300.top AND pnsOn.top AND nu_On.top AND mvOff.top  THEN
          runphase(nu1Off);
          runphase(nu2Off);

          resetAiProtection(protections.dPmaslo_gaz);
          resetDiProtection(protections.dPmaslo_gaz_less100);

          runAiProtection(protections.Pgaza_na_vyhode_nagnetatelia_GPA_STOP);
          runAiProtection(protections.Pgaza_na_vhode_nagnetatelia_GPA_STOP);
          algoritms.autoNu.CanRun:=FALSE;
          AutoNU_Off.top:=TRUE;
          (*algoritms.autoNu_1.reset(); кого, чего куда*)
      END_IF;

      IF nu1Off.top THEN
          IF (*NOT algManager.reg_V AND кто чего*) NOT pnsoff.start THEN
              runPhase(timer600);
          END_IF;
          (*IF NOT pnsoff.start THEN
              sbrosVibeg.ask();
          END_IF; kto chego?*)
      END_IF;

      IF timer600.top (*OR sbrosVibeg.answer=Answers.ANS_YES kto chto *)THEN
  	runPhase(pnsOff);
  	resetAiProtection(protections.Pmaslo_sm_nizkoe);
  	resetAiProtection(protections.Pmaslo_sm_vysokoe);
  	(*sbrosVibeg.reset (); pomogite *)
  	resetPhase(timer600);
  	(*algoritms.F2_Ch.autoAVOM_canrun_flag:=FALSE;
  	algoritms.F2_R.autoAVOM_canrun_flag:=FALSE;*)
      END_IF;
      IF (*(NOT algoritms.F2_Ch.autoAVOM_canrun_flag) AND (NOT algoritms.F2_R.autoAVOM_canrun_flag) AND*)pnsoff.start THEN
  	runPhase(Avom1Off);
  	runPhase(Avom2Off);
  	runPhase(Avom3Off);
  	runPhase(Avom4Off);

  	(*algoritms.R_AutoAVOM.CanRun:=FALSE;
  	algoritms.R_AutoAVOM.reset();
  	algoritms.S_AutoAVOM.CanRun:=FALSE;
  	algoritms.S_AutoAVOM.reset();
  	algoritms.Auto_Avom_.CanRun:=FALSE;*)
  	runPhase(autoAVOMOff);
      END_IF;

      IF pnsOff.top AND Avom1Off.top AND Avom2Off.top AND Avom3Off.top AND Avom4Off.top AND autoAVOMOff.top  THEN
          runPhase(timer5);
      END_IF;

      IF timer5.top THEN
  	resetPhase(timer5);
      END_IF;
  END_IF;

  _sunpackerCommand(command := StrAlg.inCommand);
  	source := _sunpackerCommand.source;
  	cmd := _sunpackerCommand.cmd;

  IF cmd <> 0 AND lastCmd <> cmd AND (((NOT StrAlg.opcCommandsDisabled) AND source > 0) OR source = 0) then
  	CASE BYTE_TO_INT(cmd) OF
  		(*cmdRun*) 1: 	IF (StrAlg.CanRun) THEN
  					StrAlg.isRuning := TRUE;
  					StrAlg.isEnded := FALSE;
  					StrAlg.hasError := FALSE;
  					(*****************       OnRun       *****************)

                                                    algManager.nMode:=ModeGpa.MODE_NO;
                                                    (*runIfNotRunningSO(IM.SingleOutputs.Lampa_NO);*)

                                                    runPhase(kran4Close);
                                                    runPhase(timer120);
                                                    runPhase(nu1Off);
                                                    runPhase(timer600);

                                                   (* resetAiProtection(protections.Pgaza_na_vyhode_nagnetatelia);
                                                    resetAiProtection(protections.dPmaslo_gaz);
                                                    resetAiProtection(protections.Pmaslo_sm_nizkoe);
                                                    resetAiProtection(protections.Pmaslo_sm_vysokoe);
                                                    resetAiProtection(protections.Pgaza_na_vhode_nagnetatelia);
                                                    resetAiProtection(protections.Pgaza_na_vyhode_nagnetatelia);
                                                    resetDiProtection(protections.Reg_vozb_off);
                                                    resetDiProtection(protections.Fail_chastotnii_pusk);*)

  					cmd_for_Status := cmd;
  					source_for_Status := source;
  					command_error_for_Status := 0;
  				ELSE
  					StrAlg.isRuning := FALSE;
  					StrAlg.isEnded := FALSE;
  					StrAlg.hasError 	:= FALSE;

  					cmd_for_Status := 0;
  					source_for_Status := source;
  					command_error_for_Status := cmd;
  				END_IF;
  		(*cmdReset*) 2: 	StrAlg.isRuning := FALSE;
  				StrAlg.isEnded := FALSE;
  				StrAlg.hasError 	:= FALSE;

                                           (*****************       OnReset       *****************)
                                          waitReset(IN:=FALSE);
                                          (*resetIfRunningSO(IM.SingleOutputs.Lampa_NO);*)
                                          resetIfRunning(algoritms.vibegPNS);
                                          (*impulseSO(Im.SingleOutputs.SbrosBREO);*)

                                          resetPhase(timer120);
                                          resetPhase(kran6Open);
                                          resetPhase(pnsOn);
                                          resetPhase(kran4Close);
                                          resetPhase(kran3bOpen);
                                          resetPhase(mvOff);
                                          resetPhase(kran1Close);
                                          resetPhase(kran2Close);
                                          resetPhase(kran3Close);
                                          resetPhase(kran5Open);
  	                              resetPhase(error_Krans);
                                          resetPhase(autoPnsOff);
                                          resetPhase(pnsOn);
                                          resetPhase(Pg_VhodLessThen300);
                                          resetPhase(Pg_VyhodLessThen300);
                                          resetPhase(nu2Off);
                                          resetPhase(nu1Off);
                                          resetPhase(AutoNU_Off);
                                          resetPhase(timer600);

  				cmd_for_Status := cmd;
  				source_for_Status := source;
  				command_error_for_Status := 0;
  	END_CASE;
  	resetCmdTimer(IN := false);
  	resetCmdTimerPriznak := TRUE;
  END_IF;
  lastCmd := cmd;

  resetCmdTimer(IN := resetCmdTimerPriznak, PT := T#5S);
  IF resetCmdTimer.Q THEN
  	resetCmdTimerPriznak := FALSE;
  	source_for_Status := 0;
  	cmd_for_Status := 0;
  	command_error_for_Status := 0;
  END_IF;

  StrAlg.Start:= timer120.startStatus
              OR kran6Open.startStatus
              OR pnsOn.startStatus
              OR kran4Close.startStatus
              OR kran3bOpen.startStatus
              OR mvOff.startStatus
              OR kran1Close.startStatus
              OR kran2Close.startStatus
              OR kran3Close.startStatus
              OR kran5Open.startStatus
              OR error_Krans.startStatus
              OR autoPnsOff.startStatus
              OR pnsOn.startStatus
              OR Pg_VhodLessThen300.startStatus
              OR Pg_VyhodLessThen300.startStatus
              OR nu2Off.startStatus
              OR nu1Off.startStatus
              OR AutoNU_Off.startStatus
              OR timer600.startStatus;

  StrAlg.Error:= timer120.errorStatus
              OR kran6Open.errorStatus
              OR pnsOn.errorStatus
              OR kran4Close.errorStatus
              OR kran3bOpen.errorStatus
              OR mvOff.errorStatus
              OR kran1Close.errorStatus
              OR kran2Close.errorStatus
              OR kran3Close.errorStatus
              OR kran5Open.errorStatus
              OR error_Krans.errorStatus
              OR autoPnsOff.errorStatus
              OR pnsOn.errorStatus
              OR Pg_VhodLessThen300.errorStatus
              OR Pg_VyhodLessThen300.errorStatus
              OR nu2Off.errorStatus
              OR nu1Off.errorStatus
              OR AutoNU_Off.errorStatus
              OR timer600.errorStatus;

  StrAlg.Top:=   timer120.topStatus
              OR kran6Open.topStatus
              OR pnsOn.topStatus
              OR kran4Close.topStatus
              OR kran3bOpen.topStatus
              OR mvOff.topStatus
              OR kran1Close.topStatus
              OR kran2Close.topStatus
              OR kran3Close.topStatus
              OR kran5Open.topStatus
              OR error_Krans.topStatus
              OR autoPnsOff.topStatus
              OR pnsOn.topStatus
              OR Pg_VhodLessThen300.topStatus
              OR Pg_VyhodLessThen300.topStatus
              OR nu2Off.topStatus
              OR nu1Off.topStatus
              OR AutoNU_Off.topStatus
              OR timer600.topStatus;

  (*TODO: TYPE PROGRAM CODE HERE*)
  StrAlg.status :=  SHL(BYTE_TO_DWORD(source_for_Status), 29)
  			OR SHL(BYTE_TO_DWORD(cmd_for_Status), 26)
  			OR SHL(BYTE_TO_DWORD(command_error_for_Status), 23)
  			OR SHL(BOOL_TO_DWORD(StrAlg.OpcCommandsDisabled ), 21)
  			OR SHL(BOOL_TO_DWORD(StrAlg.hasError),4)
  			OR SHL(BOOL_TO_DWORD(StrAlg.CanRun),2)
  			OR SHL(BOOL_TO_DWORD(StrAlg.isEnded),1)
  			OR BOOL_TO_DWORD(StrAlg.isRuning);
END_FUNCTION_BLOCK

FUNCTION_BLOCK AOAlg
  VAR_IN_OUT
    StrAlg : struct_Alg;
  END_VAR
  VAR
    kran6Open : struct_PhaseAlgoritm;
    kran4Close : struct_PhaseAlgoritm;
    kran3bOpen : struct_PhaseAlgoritm;
    mvOff : struct_PhaseAlgoritm;
    kran1Close : struct_PhaseAlgoritm;
    kran2Close : struct_PhaseAlgoritm;
    kran3Close : struct_PhaseAlgoritm;
    kran5Open : struct_PhaseAlgoritm;
    autoPnsOff : struct_PhaseAlgoritm;
    pnsOn : struct_PhaseAlgoritm;
    Pg_VhodLessThen300 : struct_PhaseAlgoritm;
    Pg_VyhodLessThen300 : struct_PhaseAlgoritm;
    nu1off : struct_PhaseAlgoritm;
    nu2off : struct_PhaseAlgoritm;
    AutoNU_Off : struct_PhaseAlgoritm;
    timer600 : struct_PhaseAlgoritm;
    pnsOff : struct_PhaseAlgoritm;
    Avom1Off : struct_PhaseAlgoritm;
    Avom2Off : struct_PhaseAlgoritm;
    Avom3Off : struct_PhaseAlgoritm;
    Avom4Off : struct_PhaseAlgoritm;
    autoAVOMOff : struct_PhaseAlgoritm;
    timer5 : struct_PhaseAlgoritm;
    klapan1 : struct_PhaseAlgoritm;
    klapan2 : struct_PhaseAlgoritm;
    nu_On : struct_PhaseAlgoritm;
    Start_AO_From : struct_PhaseAlgoritm;
    fb_kran6Open : fb_ph_Kran;
    fb_pnsOn : fb_ph_Switch;
    fb_kran4Close : fb_ph_Kran;
    fb_kran3bOpen : fb_ph_Kran;
    fb_mvOff : fb_ph_SectionSwitch;
    fb_kran1Close : fb_ph_Kran;
    fb_kran2Close : fb_ph_Kran;
    fb_kran3Close : fb_ph_Kran;
    fb_kran5Open : fb_ph_Kran;
    fb_autoPnsOff : fb_ph_algoritm;
    fb_Pg_VhodLessThen300 : fb_ph_CustomPhase;
    fb_Pg_VyhodLessThen300 : fb_ph_CustomPhase;
    fb_nu1Off : fb_ph_OilPump;
    fb_nu2Off : fb_ph_OilPump;
    fb_autoNuOff : fb_ph_algoritm;
    fb_timer600 : fb_ph_Timer;
    fb_pnsOff : fb_ph_Switch;
    fb_Avom1Off : fb_ph_Switch;
    fb_Avom2Off : fb_ph_Switch;
    fb_Avom3Off : fb_ph_Switch;
    fb_Avom4Off : fb_ph_Switch;
    fb_autoAVOMOff : fb_ph_algoritm;
    fb_timer5 : fb_ph_Timer;
    fb_klapan1 : fb_ph_CustomPhase;
    fb_klapan2 : fb_ph_CustomPhase;
    fb_nu_On : fb_ph_CustomPhase;
    fb_Start_AO_From : fb_ph_CustomPhase;
    _sunpackerCommand : fb_sunpackerCommand;
    _statusAi : TYPE_StatusAi;
    _Answers : TYPE_Answers;
    _statusDualInput : TYPE_statusDualInput;
    _commandDualInput : TYPE_commandDualInput;
    _DualStateImAction : TYPE_DualStateImAction;
    _PhaseAlgoritmAction : TYPE_PhaseAlgoritmAction;
    source : BYTE;
    cmd : BYTE;
    lastCmd : BYTE;
    source_for_Status : BYTE;
    cmd_for_Status : BYTE;
    command_error_for_Status : BYTE;
    resetCmdTimer : TON;
    resetCmdTimerPriznak : BOOL;
    onInit : BOOL;
    waitReset : TON;
  END_VAR
  VAR_EXTERNAL
    IM : ImConfig;
    algoritms : AlgoritmsConfig;
    ai : AiConfig;
    protections : ProtectionsConfig;
    ModeGpa : TYPE_ModeGpa;
    algManager : struct_AlgoritmsManager;
    AlgTimers : struct_AlgTimers;
  END_VAR
  VAR CONSTANT
    Ust_Pgaza : LREAL      := 0.3;
  END_VAR

  IF NOT onInit THEN
      fb_kran6Open(phaseNumber:=1, act:=_on);
      fb_kran4Close(phaseNumber:=2, act:=_off);
      fb_kran3bOpen(phaseNumber:=3, act:=_off);
      fb_mvOff(phaseNumber:=4, act:=_off);
      fb_kran1Close(phaseNumber:=5, act:=_off);
      fb_kran2Close(phaseNumber:=6, act:=_off);
      fb_kran3Close(phaseNumber:=7, act:=_off);
      fb_kran5Open(phaseNumber:=8, act:=_on);
      fb_autoPnsOff(phaseNumber:=9, act:=_reset, waitCompletion:=FALSE);
      fb_pnsOn(phaseNumber:=10, act:=_on);
      fb_Pg_VhodLessThen300(phaseNumber:=11);
      fb_Pg_VyhodLessThen300(phaseNumber:=12);
      fb_nu1Off(phaseNumber:=13, act:=_off);
      fb_nu2Off(phaseNumber:=14, act:=_off);
      fb_autoNuOff(phaseNumber:=15, act:=_reset, waitCompletion:=FALSE);
      fb_timer600(phaseNumber:=16, delay:=T#600S);
      fb_pnsOff(phaseNumber:=17, act:=_off);
      fb_Avom1Off(phaseNumber:=18, act:=_off);
      fb_Avom2Off(phaseNumber:=19, act:=_off);
      fb_Avom3Off(phaseNumber:=20, act:=_off);
      fb_Avom4Off(phaseNumber:=21, act:=_off);
      fb_autoAVOMOff(phaseNumber:=22, act:=_reset, waitCompletion:=FALSE);
      fb_timer5(phaseNumber:=23, delay:=T#5S);
      fb_klapan1(phaseNumber:=24);
      fb_klapan2(phaseNumber:=25);
      fb_nu_On(phaseNumber:=26);
      fb_Start_AO_From(phaseNumber:=27);
  onInit:=TRUE;
  END_IF;

  fb_kran6Open(StrPh:=kran6Open, Im:=Im.kran6);
  fb_pnsOn(StrPh:=pnsOn, Im:=Im.pns);
  fb_kran4Close(StrPh:=kran4Close, Im:=Im.kran4);
  fb_kran3bOpen(StrPh:=kran3bOpen, Im:=Im.kran3b);
  fb_mvOff(StrPh:=mvOff, Im:=Im.mv);
  fb_kran1Close(StrPh:=kran1Close, Im:=Im.kran1);
  fb_kran2Close(StrPh:=kran2Close, Im:=Im.Kran2);
  fb_kran3Close(StrPh:=kran3Close, Im:=Im.Kran3);
  fb_kran5Open(StrPh:=kran5Open, Im:=Im.Kran5);
  fb_autoPnsOff(StrPh:=autoPnsOff, alg:=algoritms.autoPns);
  fb_Pg_VhodLessThen300(StrPh:=Pg_VhodLessThen300);
  fb_Pg_VyhodLessThen300(StrPh:=Pg_VyhodLessThen300);
  fb_nu1Off(StrPh:=nu1off, Im:=Im.nu1);
  fb_nu2Off(StrPh:=nu2off, Im:=Im.nu2);
  fb_autoNuOff(StrPh:=AutoNU_Off, alg:=algoritms.autoNu);
  fb_timer600(StrPh:=timer600, timer:=AlgTimers.No_wait600);
  fb_pnsOff(StrPh:=pnsOff, Im:=Im.pns);
  fb_Avom1Off(StrPh:=Avom1Off, Im:=Im.v1_Avom);
  fb_Avom2Off(StrPh:=Avom2Off, Im:=Im.v2_Avom);
  fb_Avom3Off(StrPh:=Avom3Off, Im:=Im.v3_Avom);
  fb_Avom4Off(StrPh:=Avom4Off, Im:=Im.v4_Avom);
  fb_autoAVOMOff(StrPh:=autoAVOMOff, alg:=algoritms.AutoAvom);
  fb_timer5(StrPh:=timer5, timer:=AlgTimers.No_wait5);
  fb_klapan1(StrPh:=klapan1);
  fb_klapan2(StrPh:=klapan2);
  fb_nu_On(StrPh:=nu_On);
  fb_Start_AO_From(StrPh:=Start_AO_From);

  StrAlg.CanRun := StrAlg.inCanRun;
  StrAlg.OpcCommandsDisabled := StrAlg.inOpcCommandsDisabled;

  IF StrAlg.isRuning THEN

      IF	(*algoritms.F3.Smazka_1_2 OR*) IM.kran1.onStatus = _statusDualInput.STATUS_ON OR IM.kran1.onStatus = _statusDualInput.STATUS_TRANSITIONAL
  	    OR IM.kran2.onStatus = _statusDualInput.STATUS_ON OR IM.kran2.onStatus = _statusDualInput.STATUS_TRANSITIONAL  THEN
  	    IF (*(algoritms.F3.Smazka_1_2 OR*) IM.kran1.onStatus = _statusDualInput.STATUS_ON OR IM.kran1.onStatus = _statusDualInput.STATUS_TRANSITIONAL AND NOT klapan1.start AND NOT kran1Close.top THEN
  		    runPhase(klapan1);
  	    END_IF;
  	    IF (*algoritms.F3.Smazka_1_2 OR*) IM.kran2.onStatus = _statusDualInput.STATUS_ON OR IM.kran2.onStatus = _statusDualInput.STATUS_TRANSITIONAL AND NOT klapan2.start AND NOT kran2Close.top THEN
  		    runPhase(klapan2);
      	END_IF;
  	(*algoritms.F3.Smazka_1_2:=FALSE; у меня нет такой штуки*)
      END_IF;

     (* IF NOT kran6Open.start THEN
  	    ystavki.Block_kr6_alg.setValue (1);
  	    IF IM.kran6._cmdreset.IN = FALSE THEN
  		    ystavki.Block_kr6_alg.setValue (0); такой штуки тоже нет
  		        runPhase(kran6Open);
  	    END_IF;
      END_IF;*)

      (*IF NOT kran4Close.start THEN
  	    ystavki.Block_kr4_alg.setValue (1);
  	    IF IM.kran4._cmdreset.IN = FALSE THEN
  		    ystavki.Block_kr4_alg.setValue (0);
  		    kran4Close.run();
  	    END_IF;
      END_IF;*)

      (*IF NOT kran3bOpen.start THEN
  	    ystavki.Block_kr3b_alg.setValue (1);
  	    IF IM.kran3b._cmdreset.IN = FALSE THEN
  		    ystavki.Block_kr3b_alg.setValue (0);
  		    runPhase(kran3bOpen);
  	    END_IF;
      END_IF;*)

      resetDiProtection(protections.mvOff);
      resetDiProtection(protections.Off_avar_vikluchatel);
      resetDiProtection(protections.Reg_vozb_off);
      resetDiProtection(protections.Kran1_sdvig);
      resetDiProtection(protections.Kran2_sdvig);
      runPhase(mvOff);

      (*IF NOT kran1Close.start THEN
  	ystavki.Block_kr1_alg.setValue (1);*)
  	    (*IF IM.kran1._cmdreset.IN = FALSE THEN
  		    ystavki.Block_kr1_alg.setValue (0);
  		    runPhase(kran1Close);
  	    END_IF;
      END_IF;*)

      (*IF NOT kran2Close.start THEN
  	    ystavki.Block_kr2_alg.setValue (1);
  	    IF IM.kran2._cmdreset.IN = FALSE THEN
  		    ystavki.Block_kr2_alg.setValue (0);
  		    runPhase(kran2Close);
  	    END_IF;
      END_IF;*)

      (*IF NOT kran3Close.start THEN
  	    ystavki.Block_kr3_alg.setValue (1);
  	    IF	IM.kran3._cmdreset.IN = FALSE THEN
  		    ystavki.Block_kr3_alg.setValue (0);
  		    runPhase(kran3Close);
  	    END_IF;
      END_IF;*)

      (*IF kran6Open.top THEN
  	    algoritms.S_Vibr.CanRun:=FALSE;
  	    algoritms.S_Vibr.reset ();
      END_IF;*)

      IF klapan1.start AND kran1Close.top THEN
  	    (*IM.Kr1_Smazka.impulse();*)
  	    klapan1.top:=TRUE;
      END_IF;
      IF	klapan2.start AND kran2Close.top THEN
  	    (*zIM.Kr2_Smazka.impulse();*)
  	    klapan2.top:=TRUE;
      END_IF;

      (*IF 	kran1Close.top AND kran2Close.top AND kran3Close.top AND kran4Close.top AND NOT kran5Open.top THEN
  	    IF	NOT	kran5Open.start THEN
              ystavki.Block_kr5_alg.setValue (1);
  		    IF	IM.kran5._cmdreset.IN = FALSE THEN
  			    ystavki.Block_kr5_alg.setValue (0);
  			    runPhase(kran5Open);
  		    END_IF;
  	    END_IF;

  	    resetAiProtection(protections.Pgaza_na_vyhode_nagnetatelia);
      END_IF; *)

      IF mvOff.top (*AND NOT flag1*) THEN
  	    (*algoritms.AutoPNS_Start.canrun :=FALSE;
  	    algoritms.AutoPNS_Start.reset ();*)
  	    algoritms.autoPns.canrun :=FALSE;
  	    runPhase(autoPnsOff);
  	    runPhase(pnsOn);
  	    runPhase(nu_On);
  	    (*vkluchit nasosi*)
  	    algoritms.autoNu.canrun:=FALSE;
  	    (*algoritms.autoNu_2.reset ();
  	    algoritms.autoNu_1.canrun:=TRUE;
  	    algoritms.autoNu_1.run ();
  	    flag1:=TRUE;*)
      END_IF;

      IF	IM.nu1.onStatus =_statusDualInput.STATUS_ON OR IM.nu2.onStatus =_statusDualInput.STATUS_ON AND nu_On.start AND NOT nu_On.top THEN
  	    nu_On.top:=TRUE;
      END_IF;

      IF kran5Open.top THEN
  	    runPhase(Pg_VhodLessThen300);
  	    runPhase(Pg_VyhodLessThen300);
  	END_IF;

      IF Pg_VhodLessThen300.start AND NOT Pg_VhodLessThen300.top THEN
  	    IF ai.Pgaza_na_vhode_nagnetatelia.interval >= _statusAi.NORMAL AND ai.Pgaza_na_vhode_nagnetatelia.value < 0.3 THEN
  		    Pg_VhodLessThen300.top:=TRUE;
  	    END_IF;
      END_IF;

      IF Pg_VyhodLessThen300.start AND NOT Pg_VyhodLessThen300.top THEN
  	    IF ai.Pgaza_na_vyhode_nagnetatelia.interval>=_statusAi.NORMAL AND ai.Pgaza_na_vyhode_nagnetatelia.value < 0.3 THEN
  		    Pg_VyhodLessThen300.top:=TRUE;
  	    END_IF;
      END_IF;

      IF Pg_VhodLessThen300.top AND Pg_VyhodLessThen300.top AND pnsOn.top AND nu_On.top AND mvOff.top THEN
  	    runPhase(nu1Off);
      	    resetAiProtection(protections.dPmaslo_gaz);
  	    resetDiProtection(protections.dPmaslo_gaz_less100);
  	    runAiProtection(protections.Pgaza_na_vhode_nagnetatelia_GPA_STOP);
  	    runAiProtection(protections.Pgaza_na_vyhode_nagnetatelia_GPA_STOP);
  	    AutoNU_Off.top:=TRUE;
      	(*algoritms.autoNu_1.CanRun:=FALSE;
  	    algoritms.autoNu_1.reset ();*)
      END_IF;

      (*IF nuOff.top THEN
  	    IF NOT algmanager.reg_V AND NOT pnsoff.start THEN
  		    runPhase(timer600);
  	    END_IF;
  	    IF	NOT pnsoff.start THEN
  		    sbrosVibeg.ask();
  	    END_IF;
      END_IF;*)

      IF timer600.top (*OR sbrosVibeg.answer=Answers.ANS_YES*)  THEN
  	    runPhase(pnsOff);
  	    resetAiProtection(protections.Pmaslo_sm_nizkoe);
  	    resetAiProtection(protections.Pmaslo_sm_vysokoe);
  	    (*resetPhase(sbrosVibeg);*)
  	    resetPhase(timer600);
  	    (*algoritms.F2_Ch.autoAVOM_canrun_flag:=FALSE;
  	    algoritms.F2_R.autoAVOM_canrun_flag:=FALSE;*)
      END_IF;

      IF (*NOT algoritms.F2_Ch.autoAVOM_canrun_flag AND NOT algoritms.F2_R.autoAVOM_canrun_flag AND*) pnsoff.start THEN
  	    runPhase(Avom1Off);
  	    runPhase(Avom2Off);
  	    runPhase(Avom3Off);
  	    runPhase(Avom4Off);
  	    (*algoritms.R_AutoAVOM.CanRun:=FALSE;
  	    algoritms.R_AutoAVOM.reset();
  	    algoritms.S_AutoAVOM.CanRun:=FALSE;
  	    algoritms.S_AutoAVOM.reset();
  	    algoritms.Auto_Avom_.CanRun:=FALSE;*)
  	    runPhase(autoAVOMOff);
      END_IF;

      IF pnsOff.top AND Avom1Off.top AND Avom2Off.top AND Avom3Off.top AND Avom4Off.top AND autoAVOMOff.top  THEN
  	    runPhase(timer5);
      END_IF;

      IF timer5.top THEN
  	    runPhase(timer5);
      END_IF;
  END_IF;

  _sunpackerCommand(command := StrAlg.inCommand);
  	source := _sunpackerCommand.source;
  	cmd := _sunpackerCommand.cmd;

  IF cmd <> 0 AND lastCmd <> cmd AND (((NOT StrAlg.opcCommandsDisabled) AND source > 0) OR source = 0) then
  	CASE BYTE_TO_INT(cmd) OF
  		(*cmdRun*) 1: 	IF (StrAlg.CanRun) THEN
  					StrAlg.isRuning := TRUE;
  					StrAlg.isEnded := FALSE;
  					StrAlg.hasError := FALSE;
  					(*****************       OnRun       *****************)

                                                    algManager.nMode:=ModeGpa.MODE_NO;
                                                    (*runIfNotRunningSO(IM.SingleOutputs.Lampa_NO);*)

                                                    runPhase(kran4Close);
                                                    (*runPhase(timer120);*)
                                                    runPhase(nu1Off);
                                                    runPhase(timer600);

                                                   (* resetAiProtection(protections.Pgaza_na_vyhode_nagnetatelia);
                                                    resetAiProtection(protections.dPmaslo_gaz);
                                                    resetAiProtection(protections.Pmaslo_sm_nizkoe);
                                                    resetAiProtection(protections.Pmaslo_sm_vysokoe);
                                                    resetAiProtection(protections.Pgaza_na_vhode_nagnetatelia);
                                                    resetAiProtection(protections.Pgaza_na_vyhode_nagnetatelia);
                                                    resetDiProtection(protections.Reg_vozb_off);
                                                    resetDiProtection(protections.Fail_chastotnii_pusk);*)

  					cmd_for_Status := cmd;
  					source_for_Status := source;
  					command_error_for_Status := 0;
  				ELSE
  					StrAlg.isRuning := FALSE;
  					StrAlg.isEnded := FALSE;
  					StrAlg.hasError 	:= FALSE;

  					cmd_for_Status := 0;
  					source_for_Status := source;
  					command_error_for_Status := cmd;
  				END_IF;
  		(*cmdReset*) 2: 	StrAlg.isRuning := FALSE;
  				StrAlg.isEnded := FALSE;
  				StrAlg.hasError 	:= FALSE;

                                           (*****************       OnReset       *****************)
                                          waitReset(IN:=FALSE);
                                          (*resetIfRunningSO(IM.SingleOutputs.Lampa_NO);*)
                                          resetIfRunning(algoritms.vibegPNS);
                                          (*impulseSO(Im.SingleOutputs.SbrosBREO);*)

                                          (*resetPhase(timer120);*)
                                          resetPhase(kran6Open);
                                          resetPhase(pnsOn);
                                          resetPhase(kran4Close);
                                          resetPhase(kran3bOpen);
                                          resetPhase(mvOff);
                                          resetPhase(kran1Close);
                                          resetPhase(kran2Close);
                                          resetPhase(kran3Close);
                                          resetPhase(kran5Open);
  	                              (*resetPhase(error_Krans);*)
                                          resetPhase(autoPnsOff);
                                          resetPhase(pnsOn);
                                          resetPhase(Pg_VhodLessThen300);
                                          resetPhase(Pg_VyhodLessThen300);
                                          resetPhase(nu2Off);
                                          resetPhase(nu1Off);
                                          resetPhase(AutoNU_Off);
                                          resetPhase(timer600);

  				cmd_for_Status := cmd;
  				source_for_Status := source;
  				command_error_for_Status := 0;
  	END_CASE;
  	resetCmdTimer(IN := false);
  	resetCmdTimerPriznak := TRUE;
  END_IF;
  lastCmd := cmd;

  resetCmdTimer(IN := resetCmdTimerPriznak, PT := T#5S);
  IF resetCmdTimer.Q THEN
  	resetCmdTimerPriznak := FALSE;
  	source_for_Status := 0;
  	cmd_for_Status := 0;
  	command_error_for_Status := 0;
  END_IF;

  StrAlg.Start:= kran6Open.startStatus
              OR pnsOn.startStatus
              OR kran4Close.startStatus
              OR kran3bOpen.startStatus
              OR mvOff.startStatus
              OR kran1Close.startStatus
              OR kran2Close.startStatus
              OR kran3Close.startStatus
              OR kran5Open.startStatus
              OR Pg_VhodLessThen300.startStatus
              OR nu1off.startStatus
              OR nu2off.startStatus
              OR Pg_VyhodLessThen300.startStatus
              OR AutoNU_Off.startStatus
              OR timer600.startStatus
              OR pnsOff.startStatus
              OR Avom1Off.startStatus
              OR Avom2Off.startStatus
              OR Avom3Off.startStatus
              OR Avom4Off.startStatus
              OR autoAVOMOff.startStatus
              OR timer5.startStatus
              OR klapan1.startStatus
              OR klapan2.startStatus
              OR nu_On.startStatus
              OR Start_AO_From.startStatus;

  StrAlg.Error:= kran6Open.errorStatus
              OR pnsOn.errorStatus
              OR kran4Close.errorStatus
              OR kran3bOpen.errorStatus
              OR mvOff.errorStatus
              OR kran1Close.errorStatus
              OR kran2Close.errorStatus
              OR kran3Close.errorStatus
              OR kran5Open.errorStatus
              OR Pg_VhodLessThen300.errorStatus
              OR nu1off.errorStatus
              OR nu2off.errorStatus
              OR Pg_VyhodLessThen300.errorStatus
              OR AutoNU_Off.errorStatus
              OR timer600.errorStatus
              OR pnsOff.errorStatus
              OR Avom1Off.errorStatus
              OR Avom2Off.errorStatus
              OR Avom3Off.errorStatus
              OR Avom4Off.errorStatus
              OR autoAVOMOff.errorStatus
              OR timer5.errorStatus
              OR klapan1.errorStatus
              OR klapan2.errorStatus
              OR nu_On.errorStatus
              OR Start_AO_From.errorStatus;

  StrAlg.Top:= kran6Open.topStatus
              OR pnsOn.topStatus
              OR kran4Close.topStatus
              OR kran3bOpen.topStatus
              OR mvOff.topStatus
              OR kran1Close.topStatus
              OR kran2Close.topStatus
              OR kran3Close.topStatus
              OR kran5Open.topStatus
              OR Pg_VhodLessThen300.topStatus
              OR nu1off.topStatus
              OR nu2off.topStatus
              OR Pg_VyhodLessThen300.topStatus
              OR AutoNU_Off.topStatus
              OR timer600.topStatus
              OR pnsOff.topStatus
              OR Avom1Off.topStatus
              OR Avom2Off.topStatus
              OR Avom3Off.topStatus
              OR Avom4Off.topStatus
              OR autoAVOMOff.topStatus
              OR timer5.topStatus
              OR klapan1.topStatus
              OR klapan2.topStatus
              OR nu_On.topStatus
              OR Start_AO_From.topStatus;

  (*TODO: TYPE PROGRAM CODE HERE*)
  StrAlg.status :=  SHL(BYTE_TO_DWORD(source_for_Status), 29)
  			OR SHL(BYTE_TO_DWORD(cmd_for_Status), 26)
  			OR SHL(BYTE_TO_DWORD(command_error_for_Status), 23)
  			OR SHL(BOOL_TO_DWORD(StrAlg.OpcCommandsDisabled ), 21)
  			OR SHL(BOOL_TO_DWORD(StrAlg.hasError),4)
  			OR SHL(BOOL_TO_DWORD(StrAlg.CanRun),2)
  			OR SHL(BOOL_TO_DWORD(StrAlg.isEnded),1)
  			OR BOOL_TO_DWORD(StrAlg.isRuning);
END_FUNCTION_BLOCK

FUNCTION nsCepeiUpravlenya : BOOL
  VAR_INPUT
    im : ImConfig;
  END_VAR

  nsCepeiUpravlenya:=
  	im.kran1.So OR im.kran1.Sz OR
  	im.kran2.So OR im.kran2.Sz OR
  	im.kran4.So OR im.kran4.Sz OR
  	im.kran5.So OR im.kran5.Sz OR
  	(*im.kran6.So OR im.kran6.Sz OR*)
  	im.kran3b.So OR im.kran3b.Sz OR
  	im.pns.breakCmdOn OR
  	im.nu1.breakCmdOn OR
  	im.nu2.breakCmdOn OR
  	im.PNS.breakCmdOn OR
            im.v1_Avom.breakCmdOn OR
            im.v2_Avom.breakCmdOn OR
            (*im.Ten.breakCmdOn OR*)
  	im.mv.breakCmdOff;
END_FUNCTION

FUNCTION anyProtectionSignaling : BOOL
  VAR_INPUT
    protections : ProtectionsConfig;
  END_VAR

  anyProtectionSignaling:=
  protections.Topornogo_podshipnika_EDT_1.Signaling OR
  protections.Toy_podshipnika_EDT_2.Signaling OR
  protections.Toy_podshipnika_kol_EDT_3.Signaling OR
  protections.Toy_podshipnika_kol_EDT_4.Signaling OR
  protections.To_podshipnika_shest_red_EDT_5.Signaling OR
  protections.To_podshipnika_shest_red_EDT_6.Signaling OR
  protections.To_podshipnika_N_EDT_7.Signaling OR
  protections.To_podshipnika_svob_konca_EDT_8.Signaling OR
  protections.Ty_podshipnika_rab_kol_EDT_9.Signaling OR
  protections.Typornogo_podshipnika_nerab_kolodok_HT_10.Signaling OR
  protections.Tgaza_na_vyhode_H.Signaling OR
  protections.Os_sdvig_nagnetatelja_plus.Signaling OR
  protections.Os_sdvig_nagnetatelja_minus.Signaling OR
  protections.Pgaza_na_vyhode_nagnetatelia_GPA_STOP.Signaling OR
  protections.Pgaza_na_vhode_nagnetatelia_GPA_STOP.Signaling OR
  protections.Pgaza_na_vyhode_nagnetatelia.Signaling OR
  protections.dPmaslo_gaz.Signaling OR
  protections.Pmaslo_sm_nizkoe.Signaling OR
  protections.Pmaslo_sm_vysokoe.Signaling OR
  protections.Vibro_skorost_OPED_T1.Signaling OR
  protections.Vibro_skorost_OPED_T2.Signaling OR
  protections.Vibro_skorost_OYP_kolesa_ED_T3.Signaling OR
  protections.Vibro_skorost_OP_kolesa_RH_T4.Signaling OR
  protections.Vibro_skorost_OP_shesterni_RED_T5.Signaling OR
  protections.Vibro_skorost_OP_shesterni_RED_T6.Signaling OR
  protections.dPmaslo_gaz_less100.Signaling OR
  protections.Reg_vozb_off.Signaling OR
  protections.Fail_chastotnii_pusk.Signaling OR
  protections.Off_avar_vikluchatel.Signaling OR
  protections.AOKC_SHKC.Signaling OR
  protections.AO_PRU.Signaling OR
  protections.AO_ot_SHU.Signaling OR
  protections.mvOff.Signaling OR
  protections.Kran1_sdvig.Signaling OR
  protections.Kran2_sdvig.Signaling OR
  protections.Tgaza_na_vyhode_H.Signaling;
END_FUNCTION

FUNCTION anyAnalogsPs : BOOL
  VAR_INPUT
    ai : AiConfig;
  END_VAR
  VAR
    statusAi : TYPE_StatusAi;
  END_VAR

  anyAnalogsPs:=
  ai.Toporno_podshipnika_EDT_1.interval= statusAi.HW OR
  ai.Toporno_podshipnika_EDT_1.interval= statusAi.LW OR
  ai.Toy_podshipnika_EDT_2.interval= statusAi.HW OR
  ai.Toy_podshipnika_kol_EDT_3.interval= statusAi.HW OR
  ai.Ty_podshipnika_red_EDT_6.interval= statusAi.HW OR
  ai.Ty_podshipnika_nagnet_EDT_7_1.interval= statusAi.HW OR
  ai.Ty_podshipnika_nagnet_EDT_7_2.interval= statusAi.HW OR
  ai.Toy_podshipnika_svobod_konca_EDT_8_1.interval= statusAi.HW OR
  ai.Toy_podshipnika_svobod_konca_EDT_8_2.interval= statusAi.HW OR
  ai.Tholodnogo_vozduha_ED_kanal_1.interval= statusAi.HW OR
  ai.Tholodnogo_vozduha_ED_kanal_2.interval= statusAi.HW OR
  ai.Tgorjachego_vozduha_ED_kanal_1.interval= statusAi.HW OR
  ai.Tgaza_na_vyhode_H.interval= statusAi.HW OR
  ai.Tmasla_MB.interval= statusAi.LW OR
  ai.Pmasla_posle_GNS.interval= statusAi.LW OR
  ai.Pmasla_posle_NU.interval= statusAi.LW OR
  ai.dPgaza_na_konfuzore.interval= statusAi.HW OR
  ai.Os_sdvig_nagnetatelja_plus.interval= statusAi.HW OR
  ai.Os_sdvig_nagnetatelja_minus.interval= statusAi.HW OR
  ai.dPmaslo_gaz.interval= statusAi.HW OR
  ai.Pgaza_na_vhode_nagnetatelia.interval= statusAi.HW OR
  ai.Pgaza_na_vyhode_nagnetatelia.interval= statusAi.HW OR
  ai.Pimpuls_gaz.interval= statusAi.HW OR
  ai.Pimpuls_gaz.interval= statusAi.LW OR
  ai.Yroven_masla_MB.interval= statusAi.HW OR
  ai.Yroven_masla_MB.interval= statusAi.LW OR
  ai.Tmasla_MB_TEN.interval= statusAi.HW OR
  ai.Tmasla_MB_TEN.interval= statusAi.LW OR
  ai.Vibro_skorost_OYP_kolesa_ED_T3.interval= statusAi.HW OR
  ai.Vibro_skorost_OYP_kolesa_ED_T3.interval= statusAi.LW OR
  ai.Vibro_skorost_OP_kolesa_RH_T4.interval= statusAi.HW OR
  ai.Vibro_skorost_OP_kolesa_RH_T4.interval= statusAi.LW;
END_FUNCTION

FUNCTION analogsNS : BOOL
  VAR_INPUT
    ai : AiConfig;
  END_VAR
  VAR
    statusAi : TYPE_StatusAi;
  END_VAR

  analogsNS:=
    ((ai.Tstali_statora_kanal_1.Interval < statusAi.Normal) AND NOT ai.Tstali_statora_kanal_1.remont)
  OR((ai.Tstali_statora_kanal_2.Interval < statusAi.Normal) AND NOT ai.Tstali_statora_kanal_2.remont)
  OR((ai.Tstali_statora_kanal_3.Interval < statusAi.Normal) AND NOT ai.Tstali_statora_kanal_3.remont)
  OR((ai.Tmedi_statora_kanal_1.Interval < statusAi.Normal) AND NOT ai.Tmedi_statora_kanal_1.remont)
  OR((ai.Tmedi_statora_kanal_2.Interval < statusAi.Normal) AND NOT ai.Tmedi_statora_kanal_2.remont)
  OR((ai.Tmedi_statora_kanal_3.Interval < statusAi.Normal) AND NOT ai.Tmedi_statora_kanal_3.remont)
  OR((ai.Toporno_podshipnika_EDT_1.Interval < statusAi.Normal) AND NOT ai.Toporno_podshipnika_EDT_1.remont)
  OR((ai.Toy_podshipnika_EDT_2.Interval < statusAi.Normal) AND NOT ai.Toy_podshipnika_EDT_2.remont)
  OR((ai.Toy_podshipnika_kol_EDT_3.Interval < statusAi.Normal) AND NOT ai.Toy_podshipnika_kol_EDT_3.remont)
  OR((ai.Toy_podshipnika_kol_EDT_4.Interval < statusAi.Normal) AND NOT ai.Toy_podshipnika_kol_EDT_4.remont)
  OR((ai.Toy_podshipnika_shest_red_EDT_5.Interval < statusAi.Normal) AND NOT ai.Toy_podshipnika_shest_red_EDT_5.remont)
  OR((ai.Ty_podshipnika_red_EDT_6.Interval < statusAi.Normal) AND NOT ai.Ty_podshipnika_red_EDT_6.remont)
  OR((ai.Ty_podshipnika_nagnet_EDT_7_1.Interval < statusAi.Normal) AND NOT ai.Ty_podshipnika_nagnet_EDT_7_1.remont)
  OR((ai.Ty_podshipnika_nagnet_EDT_7_2.Interval < statusAi.Normal) AND NOT ai.Ty_podshipnika_nagnet_EDT_7_2.remont)
  OR((ai.Toy_podshipnika_svobod_konca_EDT_8_1.Interval < statusAi.Normal) AND NOT ai.Toy_podshipnika_svobod_konca_EDT_8_1.remont)
  OR((ai.Toy_podshipnika_svobod_konca_EDT_8_2.Interval < statusAi.Normal) AND NOT ai.Toy_podshipnika_svobod_konca_EDT_8_2.remont)
  OR((ai.Tholodnogo_vozduha_ED_kanal_1.Interval < statusAi.Normal) AND NOT ai.Tholodnogo_vozduha_ED_kanal_1.remont)
  OR((ai.Tholodnogo_vozduha_ED_kanal_2.Interval < statusAi.Normal) AND NOT ai.Tholodnogo_vozduha_ED_kanal_2.remont)
  OR((ai.Tgorjachego_vozduha_ED_kanal_1.Interval < statusAi.Normal) AND NOT ai.Tgorjachego_vozduha_ED_kanal_1.remont)
  OR((ai.Tgorjachego_vozduha_ED_kanal_2.Interval < statusAi.Normal) AND NOT ai.Tgorjachego_vozduha_ED_kanal_2.remont)
  OR((ai.Tnarujnogo_vozduha.Interval < statusAi.Normal) AND NOT ai.Tnarujnogo_vozduha.remont)
  OR((ai.Tgaza_na_vhode_H.Interval < statusAi.Normal) AND NOT ai.Tgaza_na_vhode_H.remont)
  OR((ai.Tgaza_na_vyhode_H.Interval < statusAi.Normal) AND NOT ai.Tgaza_na_vyhode_H.remont)
  OR((ai.Tmasla_posle_AVOM.Interval < statusAi.Normal) AND NOT ai.Tmasla_posle_AVOM.remont)
  OR((ai.Tgorjachego_vozduha_ED_kanal_2.Interval < statusAi.Normal) AND NOT ai.Tgorjachego_vozduha_ED_kanal_2.remont)
  OR((ai.Tmasla_MB.Interval < statusAi.Normal) AND NOT ai.Tmasla_MB.remont)
  OR((ai.dPgaza_na_konfuzore.Interval < statusAi.Normal) AND NOT ai.dPgaza_na_konfuzore.remont)
  OR((ai.Pmaslo_sm_nizkoe.Interval < statusAi.Normal) AND NOT ai.Pmaslo_sm_nizkoe.remont)
  OR((ai.dPgaza_na_maslo_filtre.Interval < statusAi.Normal) AND NOT ai.dPgaza_na_maslo_filtre.remont)
  OR((ai.Pmaslo_sm_vysokoe.Interval < statusAi.Normal) AND NOT ai.Pmaslo_sm_vysokoe.remont)
  OR((ai.Pmasla_posle_GNS.Interval < statusAi.Normal) AND NOT ai.Pmasla_posle_GNS.remont)
  OR((ai.Pmasla_posle_NU.Interval < statusAi.Normal) AND NOT ai.Pmasla_posle_NU.remont)
  OR((ai.Os_sdvig_nagnetatelja_plus.Interval < statusAi.Normal) AND NOT ai.Os_sdvig_nagnetatelja_plus.remont)
  OR((ai.Os_sdvig_nagnetatelja_minus.Interval < statusAi.Normal) AND NOT ai.Os_sdvig_nagnetatelja_minus.remont)
  OR((ai.dPmaslo_gaz.Interval < statusAi.Normal) AND NOT ai.dPmaslo_gaz.remont)
  OR((ai.Pgaza_na_vhode_nagnetatelia.Interval < statusAi.Normal) AND NOT ai.Pgaza_na_vhode_nagnetatelia.remont)
  OR((ai.Pgaza_na_vyhode_nagnetatelia.Interval < statusAi.Normal) AND NOT ai.Pgaza_na_vyhode_nagnetatelia.remont)
  OR((ai.Pimpuls_gaz.Interval < statusAi.Normal) AND NOT ai.Pimpuls_gaz.remont)
  OR((ai.Yroven_masla_MB.Interval < statusAi.Normal) AND NOT ai.Yroven_masla_MB.remont)
  OR((ai.Kontrol_per_220V.Interval < statusAi.Normal) AND NOT ai.Kontrol_per_220V.remont)
  OR((ai.Kontrol_post_220V.Interval < statusAi.Normal) AND NOT ai.Kontrol_post_220V.remont)
  OR((ai.Kontrol_post_220V.Interval < statusAi.Normal) AND NOT ai.Kontrol_post_220V.remont)
  OR((ai.Vibro_skorost_OPED_T1.Interval < statusAi.Normal) AND NOT ai.Vibro_skorost_OPED_T1.remont)
  OR((ai.Vibro_skorost_OYP_kolesa_ED_T3.Interval < statusAi.Normal) AND NOT ai.Vibro_skorost_OYP_kolesa_ED_T3.remont)
  OR((ai.Vibro_skorost_OP_kolesa_RH_T4.Interval < statusAi.Normal) AND NOT ai.Vibro_skorost_OP_kolesa_RH_T4.remont);
END_FUNCTION

FUNCTION_BLOCK ppuAlg
  VAR_IN_OUT
    StrAlg : struct_Alg;
  END_VAR
  VAR
    BMP_Err : struct_PhaseAlgoritm;
    Level_masla_Norm : struct_PhaseAlgoritm;
    T_masla_Norm : struct_PhaseAlgoritm;
    Krans_ready_to_move : struct_PhaseAlgoritm;
  END_VAR
  VAR_IN_OUT
    Krans_Poloj : struct_PhaseAlgoritm;
    Net_AO_KC_SHKS04M : struct_PhaseAlgoritm;
    EGPA_Stop : struct_PhaseAlgoritm;
    Avt_SHU_vkl : struct_PhaseAlgoritm;
    All_IM_Off : struct_PhaseAlgoritm;
    Nalichie220_SHU_Ai : struct_PhaseAlgoritm;
    BP_Norm : struct_PhaseAlgoritm;
    Naprajenie_U_IM : struct_PhaseAlgoritm;
    MV_Poloj_RolledON : struct_PhaseAlgoritm;
    MV_Poloj_RolledOFF : struct_PhaseAlgoritm;
    NOTAnalogNS : struct_PhaseAlgoritm;
    Net_ASPS_Analogs : struct_PhaseAlgoritm;
    Not_AS : struct_PhaseAlgoritm;
    Gotov_Vozb : struct_PhaseAlgoritm;
    Reactornyi_P : struct_PhaseAlgoritm;
    Chastotnyi_P : struct_PhaseAlgoritm;
    dP_kr1 : struct_PhaseAlgoritm;
    Auto_Rej : struct_PhaseAlgoritm;
    CK_IM_Norm : struct_PhaseAlgoritm;
    HAnd_Mode : struct_PhaseAlgoritm;
    Impuls_Gaz : struct_PhaseAlgoritm;
  END_VAR
  VAR
    fb_BMP_Err : fb_ph_CustomPhase;
    fb_Level_masla_Norm : fb_ph_CustomPhase;
    fb_T_masla_Norm : fb_ph_CustomPhase;
    fb_Krans_ready_to_move : fb_ph_CustomPhase;
    fb_Krans_Poloj : fb_ph_CustomPhase;
    fb_Net_AO_KC_SHKS04M : fb_ph_CustomPhase;
    fb_EGPA_Stop : fb_ph_CustomPhase;
    fb_Avt_SHU_vkl : fb_ph_CustomPhase;
    fb_All_IM_Off : fb_ph_CustomPhase;
    fb_Nalichie220_SHU_Ai : fb_ph_CustomPhase;
    fb_BP_Norm : fb_ph_CustomPhase;
    fb_Naprajenie_U_IM : fb_ph_CustomPhase;
    fb_MV_Poloj_RolledON : fb_ph_CustomPhase;
    fb_MV_Poloj_RolledOFF : fb_ph_CustomPhase;
    fb_NOTAnalogNS : fb_ph_CustomPhase;
    fb_Net_ASPS_Analogs : fb_ph_CustomPhase;
    fb_Not_AS : fb_ph_CustomPhase;
    fb_Gotov_Vozb : fb_ph_CustomPhase;
    fb_Reactornyi_P : fb_ph_CustomPhase;
    fb_Chastotnyi_P : fb_ph_CustomPhase;
    fb_dP_kr1 : fb_ph_CustomPhase;
    fb_Auto_Rej : fb_ph_CustomPhase;
    fb_CK_IM_Norm : fb_ph_CustomPhase;
    fb_HAnd_Mode : fb_ph_CustomPhase;
    fb_Impuls_Gaz : fb_ph_CustomPhase;
    _sunpackerCommand : fb_sunpackerCommand;
    modeR_Trig : R_TRIG;
    modeF_Trig : F_TRIG;
    _statusAi : TYPE_StatusAi;
    _Answers : TYPE_Answers;
    _statusDualInput : TYPE_statusDualInput;
    _DualStateImAction : TYPE_DualStateImAction;
    _PhaseAlgoritmAction : TYPE_PhaseAlgoritmAction;
    _basketStats : TYPE_basketStats;
  END_VAR
  VAR_OUTPUT
    puskAllowed : BOOL;
    testAllowed : BOOL;
  END_VAR
  VAR
    ppuDone : BOOL;
    source : BYTE;
    cmd : BYTE;
    lastCmd : BYTE;
    source_for_Status : BYTE;
    cmd_for_Status : BYTE;
    command_error_for_Status : BYTE;
    resetCmdTimer : TON;
    resetCmdTimerPriznak : BOOL;
    onInit : BOOL;
  END_VAR
  VAR_EXTERNAL
    IM : ImConfig;
    ai : AiConfig;
    di : DiConfig;
    algManager : struct_AlgoritmsManager;
    protectManager : struct_ProtectionsManager;
    NotHasRezervNU : BOOL;
    ModeGpa : TYPE_ModeGpa;
    algoritms : AlgoritmsConfig;
  END_VAR

  IF NOT onInit THEN

      fb_BMP_Err(phaseNumber:=0);
      fb_Level_masla_Norm(phaseNumber:=1);
      fb_T_masla_Norm(phaseNumber:=2);
      fb_Krans_ready_to_move(phaseNumber:=5);
      fb_Krans_Poloj(phaseNumber:=6);
      fb_Net_AO_KC_SHKS04M(phaseNumber:=7);
      fb_EGPA_Stop(phaseNumber:=9);
      fb_Avt_SHU_vkl(phaseNumber:=10);
      fb_All_IM_Off(phaseNumber:=11);
      fb_Nalichie220_SHU_Ai(phaseNumber:=12);
      fb_BP_Norm(phaseNumber:=13);
      fb_Naprajenie_U_IM(phaseNumber:=14);
      fb_MV_Poloj_RolledON(phaseNumber:=15);
      fb_MV_Poloj_RolledOFF(phaseNumber:=16);
      fb_NOTAnalogNS(phaseNumber:=17);
      fb_Net_ASPS_Analogs(phaseNumber:=18);
      fb_Not_AS(phaseNumber:=19);
      fb_Gotov_Vozb(phaseNumber:=20);
      fb_Reactornyi_P(phaseNumber:=21);
      fb_Chastotnyi_P(phaseNumber:=22);
      fb_dP_kr1(phaseNumber:=23);
      fb_Auto_Rej(phaseNumber:=24);
      fb_CK_IM_Norm(phaseNumber:=25);
      fb_HAnd_Mode(phaseNumber:=26);
      fb_Impuls_Gaz(phaseNumber:=27);

  onInit:=TRUE;
  END_IF;

  fb_BMP_Err(StrPh:=BMP_Err);
  fb_Level_masla_Norm(StrPh:=Level_masla_Norm);
  fb_T_masla_Norm(StrPh:=T_masla_Norm);
  fb_Krans_ready_to_move(StrPh:=Krans_ready_to_move);
  fb_Krans_Poloj(StrPh:=Krans_Poloj);
  fb_Net_AO_KC_SHKS04M(StrPh:=Net_AO_KC_SHKS04M);
  fb_EGPA_Stop(StrPh:=EGPA_Stop);
  fb_Avt_SHU_vkl(StrPh:=Avt_SHU_vkl);
  fb_All_IM_Off(StrPh:=All_IM_Off);
  fb_Nalichie220_SHU_Ai(StrPh:=Nalichie220_SHU_Ai);
  fb_BP_Norm(StrPh:=BP_Norm);
  fb_Naprajenie_U_IM(StrPh:=Naprajenie_U_IM);
  fb_MV_Poloj_RolledON(StrPh:=MV_Poloj_RolledON);
  fb_MV_Poloj_RolledOFF(StrPh:=MV_Poloj_RolledOFF);
  fb_NOTAnalogNS(StrPh:=NOTAnalogNS);
  fb_Net_ASPS_Analogs(StrPh:=Net_ASPS_Analogs);
  fb_Not_AS(StrPh:=Not_AS);
  fb_Gotov_Vozb(StrPh:=Gotov_Vozb);
  fb_Reactornyi_P(StrPh:=Reactornyi_P);
  fb_Chastotnyi_P(StrPh:=Chastotnyi_P);
  fb_dP_kr1(StrPh:=dP_kr1);
  fb_Auto_Rej(StrPh:=Auto_Rej);
  fb_CK_IM_Norm(StrPh:=CK_IM_Norm);
  fb_HAnd_Mode(StrPh:=HAnd_Mode);
  fb_Impuls_Gaz(StrPh:=Impuls_Gaz);

  IF StrAlg.isRuning THEN

      (*BMP_Err.top:= ((BMPERR_k = 0) OR (kontroller.imit)); надо разобраться кто такой BMPERR_k*)
      (*уровень масла в норме*)
      Level_masla_Norm.top := (ai.Yroven_masla_MB.interval = _statusAi.normal);

      (*температура масла в норме*)
      T_masla_Norm.top:= (ai.Tmasla_MB.interval = _statusAi.normal);

      (*kраны готовы к управлению*)
      Krans_ready_to_move.top:= NOT (IM.Kran1.So OR IM.Kran1.Sz OR IM.Kran2.So OR IM.Kran2.Sz OR IM.Kran3.So OR
                                     IM.Kran3.Sz OR IM.Kran3b.So OR IM.Kran3b.Sz OR IM.Kran4.So OR IM.Kran4.Sz OR
  			     IM.Kran5.So OR IM.Kran5.Sz OR IM.Kran6.So OR IM.Kran6.Sz);

      (*положение кранов верное*)
      Krans_Poloj.top:= (Im.Kran1.onStatus=_statusDualInput.STATUS_OFF) AND
  		  (Im.Kran2.onStatus=_statusDualInput.STATUS_OFF) AND
  		  (Im.Kran3.onStatus=_statusDualInput.STATUS_OFF) AND
  		  (Im.Kran3b.onStatus=_statusDualInput.STATUS_ON) AND
  		  (Im.Kran4.onStatus=_statusDualInput.STATUS_OFF) AND
  		  (Im.Kran5.onStatus=_statusDualInput.STATUS_ON) AND
                        (Im.Kran6.onStatus=_statusDualInput.STATUS_ON);
      (*Нет АО от ШКС
      Net_AO_KC_SHKS04M.top:= haveAlarms(); кто такой haveAlarms*)

      (*Режим ЭГПА остановлен *)
      EGPA_Stop.top := (algManager.mode = ModeGpa.MODE_STOP);

      (*Автомат ШУ включен *)
      Avt_SHU_vkl.top := IM.SingleSignals.SHU_v_GPA_vkluch.Q;

      (*Все исполнительные механизмы выключены *)
      All_IM_Off.top := (IM.mv.onStatus=_statusDualInput.STATUS_OFF) AND (IM.pns.onStatus=_statusDualInput.STATUS_OFF) AND
                        (IM.nu1.onStatus=_statusDualInput.STATUS_OFF) AND (IM.nu2.onStatus=_statusDualInput.STATUS_OFF) AND
                        (IM.v1_Avom.onStatus=_statusDualInput.STATUS_OFF) AND (IM.v2_Avom.onStatus=_statusDualInput.STATUS_OFF) AND
  		  (IM.v3_Avom.onStatus=_statusDualInput.STATUS_OFF)AND (IM.v4_Avom.onStatus=_statusDualInput.STATUS_OFF) AND
                        (IM.CMN.onStatus=_statusDualInput.STATUS_OFF) AND (IM.TEN_MB.onStatus=_statusDualInput.STATUS_OFF) AND
                        (IM.TEN_kollectora.onStatus=_statusDualInput.STATUS_OFF) AND (IM.KaloriferAVOM.onStatus=_statusDualInput.STATUS_OFF);

      (*Наличие 220 в шу*)
      Nalichie220_SHU_Ai.top :=	(ai.Kontrol_per_220V.interval = _statusAi.normal)	 AND (ai.Kontrol_post_220V.interval = _statusAi.normal);

      (*Блоки питания норм*)
      BP_Norm.top:=
  		(IM.SingleSignals.Nalichie_BP1.Q AND
  		IM.SingleSignals.Nalichie_BP2.Q AND
  		IM.SingleSignals.Nalichie_BP3.Q AND
  		IM.SingleSignals.Nalichie_BP4.Q AND
  		IM.SingleSignals.Nalichie_BP5.Q AND
  		IM.SingleSignals.Nalichie_BP6.Q AND
  		IM.SingleSignals.Nalichie_BP7_BP8.Q AND
  		IM.SingleSignals.Nalichie_BP9_BP10.Q AND

  		IM.SingleSignals.Nalichie_220BEAO.Q AND
  		IM.SingleSignals.Nalichie_per_220_na_vhode.Q AND
  		IM.SingleSignals.Nalichie_post_220_na_vhode.Q AND
  		IM.SingleSignals.Nalichie_BP11.Q AND
  		IM.SingleSignals.Nalichie_BP12.Q);

      (*Напряжение исполнительниых механизмов
      Naprajenie_U_IM.top := IM.NalichieU_CMN.q AND IM.NalichieU_NU1.Q AND IM.Nalichie_CU_MV.Q  AND IM.NalichieU_NU2.Q AND
  						IM.NalichieU_PNS.Q; нет сигналов таких *)

      (* положение тележки мв вкачена *)
      MV_Poloj_RolledON.top:= IM.mv.basketStatus = _basketStats.BASKET_ROLLEDIN;

      (* положение тележки мв выкачена *)
      MV_Poloj_RolledOFF.top:= IM.mv.basketStatus = _basketStats.BASKET_ROLLEDOUT;

      (* нет неисправных аналоговых сигналов *)
      NOTAnalogNS.top :=  NOT analogsNS();

      (* нет аварийных/предупредительных сигнализаций аналоговых сигналов *)
      Net_ASPS_Analogs.top := anyAnalogsPs(); (*Не понял где посмотреть наличие ас аналогов *)

      (* нет сработанных защит *)
      Not_AS.top := NOT anyProtectionSignaling();

      (* готовность возбудителя *)
      Gotov_Vozb.top:= IM.SingleSignals.Vozbud_gotovnost.Q;

      (* реакторный пуск *)
      (*Reactornyi_P.top := IM.SingleSignals.Reaktornii_pusk_perek.Q AND NOT IM.SingleSignals.Chastotny_pusk.Q;*)

      (* частотный пуск *)
     (* Chastotnyi_P.top:=IM.SingleSignals.Chastotny_pusk.Q AND NOT IM.SingleSignals.Reaktornii_pusk_perek.Q;*)

      (* нет перепада давления на кране 1 *)
      dP_kr1.top:= NOT IM.SingleSignals.dp_kran1_Less100.Q (*AND (IM.PerepadDavlenieKran1_CK.status = 1))*);

      (* в автоматическом ли режиме исполнительные механизмы *)
      (*Auto_Rej.top := im.NU1_Automat.Q AND im.PNS_Automat.Q AND im.NU2_Automat.Q;*)

      (* есть наряжение в цепях управления ИМ *)
      CK_IM_Norm.top := nsCepeiUpravlenya();

      (* ручной режим *)
      HAnd_Mode.top:= NOT im.SingleSignals.Rezhim_ruchnogo_regulirovaniya.Q;

      (* импульсный газ *)
      Impuls_Gaz.top:= ai.Pimpuls_gaz.interval=_statusAi.normal;

      ppuDone := BMP_Err.top AND
  	     Level_masla_Norm.top AND
                 T_masla_Norm.top AND
  	     Krans_ready_to_move.top AND
  	     Krans_Poloj.top AND
  	     Net_AO_KC_SHKS04M.top AND
  	     EGPA_Stop.top AND
                 Avt_SHU_vkl.top AND
                 All_IM_Off.top AND
                 Nalichie220_SHU_Ai.top AND
                 BP_Norm.top AND
                 Naprajenie_U_IM.top AND
                 MV_Poloj_RolledON.top AND
                 MV_Poloj_RolledOFF.top AND
                 NOTAnalogNS.top AND
                 Net_ASPS_Analogs.top AND
                 Not_AS.top AND
                 Gotov_Vozb.top AND
                 Reactornyi_P.top AND
                 Chastotnyi_P.top AND
                 dP_kr1.top AND
                 Auto_Rej.top AND
                 CK_IM_Norm.top AND
                 HAnd_Mode.top AND
                 Impuls_Gaz.top;

      puskAllowed:= ppuDone AND Im.mv.basketStatus = _basketStats.BASKET_ROLLEDIN;
      testAllowed:= ppuDone AND Im.mv.basketStatus = _basketStats.BASKET_ROLLEDOUT;

      modeR_Trig(CLK:=puskAllowed);
      modeF_Trig(CLK:=puskAllowed);

      IF modeR_Trig.Q THEN
  	algManager.nMode:= ModeGpa.MODE_READY;
      END_IF;
      IF modeF_Trig.Q THEN
  	algManager.nMode:= ModeGpa.MODE_STOP;
      END_IF;

      IF puskAllowed THEN
          algoritms.Apusk.inCanRun:= TRUE;
          algoritms.SemiAutoPusk.inCanRun:= TRUE;
      ELSE
          algoritms.Apusk.inCanRun:= FALSE;
          algoritms.SemiAutoPusk.inCanRun:= FALSE;
      END_IF;

      IF testAllowed THEN
          algoritms.testPms.inCanRun:=  TRUE;
          algoritms.testdPmg.inCanRun:= TRUE;
          algoritms.puskK.inCanRun:=    TRUE;
          algoritms.puskV.inCanRun:=    TRUE;
      ELSE
          algoritms.testPms.inCanRun:=  FALSE;
          algoritms.testdPmg.inCanRun:= FALSE;
          algoritms.puskK.inCanRun:=    FALSE;
          algoritms.puskV.inCanRun:=    FALSE;
      END_IF;

  END_IF;

  StrAlg.CanRun := StrAlg.inCanRun;
  StrAlg.OpcCommandsDisabled := StrAlg.inOpcCommandsDisabled;

  (* ---- Если управление с ВУ заблокировано, то  передаем команду из алгоритма ---- *)
  IF StrAlg.inOpcCommandsDisabled THEN
  	StrAlg.inCommand := StrAlg.inCommand_Alg;
  ELSE (* иначе передаем команду с АРМа*)
  	StrAlg.inCommand := StrAlg.inCommand_ARM;
  END_IF;

  _sunpackerCommand(command := StrAlg.inCommand);
  	source := _sunpackerCommand.source;
  	cmd := _sunpackerCommand.cmd;

  IF cmd <> 0 AND lastCmd <> cmd AND (((NOT StrAlg.opcCommandsDisabled) AND source > 0) OR source = 0) then
  	CASE BYTE_TO_INT(cmd) OF
  		(*cmdRun*) 1: 	IF (StrAlg.CanRun) THEN
  					StrAlg.isRuning := TRUE;
  					StrAlg.isEnded := FALSE;
  					StrAlg.hasError := FALSE;
  					(*****************       OnRun       *****************)

  					cmd_for_Status := cmd;
  					source_for_Status := source;
  					command_error_for_Status := 0;
  				ELSE
  					StrAlg.isRuning := FALSE;
  					StrAlg.isEnded := FALSE;
  					StrAlg.hasError 	:= FALSE;

  					cmd_for_Status := 0;
  					source_for_Status := source;
  					command_error_for_Status := cmd;
  				END_IF;
  		(*cmdReset*) 2: 	StrAlg.isRuning := FALSE;
  				StrAlg.isEnded := FALSE;
  				StrAlg.hasError 	:= FALSE;

                                           (*****************       OnReset       *****************)

                                                    resetPhase(BMP_Err);
                                                    resetPhase(Level_masla_Norm);
                                                    resetPhase(T_masla_Norm);
                                                    resetPhase(Krans_ready_to_move);
                                                    resetPhase(Krans_Poloj);
                                                    resetPhase(Net_AO_KC_SHKS04M);
                                                    resetPhase(EGPA_Stop);
                                                    resetPhase(Avt_SHU_vkl);
                                                    resetPhase(All_IM_Off);
                                                    resetPhase(Nalichie220_SHU_Ai);
                                                    resetPhase(BP_Norm);
                                                    resetPhase(Naprajenie_U_IM);
                                                    resetPhase(MV_Poloj_RolledON);
                                                    resetPhase(MV_Poloj_RolledOFF);
                                                    resetPhase(NOTAnalogNS);
                                                    resetPhase(Net_ASPS_Analogs);
                                                    resetPhase(Not_AS);
                                                    resetPhase(Gotov_Vozb);
                                                    resetPhase(Reactornyi_P);
                                                    resetPhase(Chastotnyi_P);
                                                    resetPhase(dP_kr1);
                                                    resetPhase(Auto_Rej);
                                                    resetPhase(CK_IM_Norm);
                                                    resetPhase(HAnd_Mode);
                                                    resetPhase(Impuls_Gaz);

                                                    algoritms.testPms.inCanRun:=  FALSE;
                                                    algoritms.testdPmg.inCanRun:= FALSE;
                                                    algoritms.puskK.inCanRun:=    FALSE;
                                                    algoritms.puskV.inCanRun:=    FALSE;

                                          StrAlg.inCanRun:=FALSE;
                                          puskAllowed:=FALSE;
                                          testAllowed:=FALSE;
                                          modeR_Trig(CLK:=FALSE);
                                          modeF_Trig(CLK:=FALSE);

  				cmd_for_Status := cmd;
  				source_for_Status := source;
  				command_error_for_Status := 0;
  	END_CASE;
  	resetCmdTimer(IN := false);
  	resetCmdTimerPriznak := TRUE;
  END_IF;
  lastCmd := cmd;

  resetCmdTimer(IN := resetCmdTimerPriznak, PT := T#5S);
  IF resetCmdTimer.Q THEN
  	resetCmdTimerPriznak := FALSE;
  	source_for_Status := 0;
  	cmd_for_Status := 0;
  	command_error_for_Status := 0;
  END_IF;

  StrAlg.Start:= BMP_Err.startStatus
              OR Level_masla_Norm.startStatus
              OR T_masla_Norm.startStatus
              OR Krans_ready_to_move.startStatus
              OR Krans_Poloj.startStatus
              OR Net_AO_KC_SHKS04M.startStatus
              OR EGPA_Stop.startStatus
              OR Avt_SHU_vkl.startStatus
              OR All_IM_Off.startStatus
              OR Nalichie220_SHU_Ai.startStatus
              OR BP_Norm.startStatus
              OR Naprajenie_U_IM.startStatus
              OR MV_Poloj_RolledON.startStatus
              OR MV_Poloj_RolledOFF.startStatus
              OR NOTAnalogNS.startStatus
              OR Net_ASPS_Analogs.startStatus
              OR Not_AS.startStatus
              OR Gotov_Vozb.startStatus
              OR Reactornyi_P.startStatus
              OR Chastotnyi_P.startStatus
              OR dP_kr1.startStatus
              OR Auto_Rej.startStatus
              OR CK_IM_Norm.startStatus
              OR HAnd_Mode.startStatus
              OR Impuls_Gaz.startStatus;

  StrAlg.Error:= BMP_Err.errorStatus
              OR Level_masla_Norm.errorStatus
              OR T_masla_Norm.errorStatus
              OR Krans_ready_to_move.errorStatus
              OR Krans_Poloj.errorStatus
              OR Net_AO_KC_SHKS04M.errorStatus
              OR EGPA_Stop.errorStatus
              OR Avt_SHU_vkl.errorStatus
              OR All_IM_Off.errorStatus
              OR Nalichie220_SHU_Ai.errorStatus
              OR BP_Norm.errorStatus
              OR Naprajenie_U_IM.errorStatus
              OR MV_Poloj_RolledON.errorStatus
              OR MV_Poloj_RolledOFF.errorStatus
              OR NOTAnalogNS.errorStatus
              OR Net_ASPS_Analogs.errorStatus
              OR Not_AS.errorStatus
              OR Gotov_Vozb.errorStatus
              OR Reactornyi_P.errorStatus
              OR Chastotnyi_P.errorStatus
              OR dP_kr1.errorStatus
              OR Auto_Rej.errorStatus
              OR CK_IM_Norm.errorStatus
              OR HAnd_Mode.errorStatus
              OR Impuls_Gaz.errorStatus;

  StrAlg.Top:=   BMP_Err.topStatus
              OR Level_masla_Norm.topStatus
              OR T_masla_Norm.topStatus
              OR Krans_ready_to_move.topStatus
              OR Krans_Poloj.topStatus
              OR Net_AO_KC_SHKS04M.topStatus
              OR EGPA_Stop.topStatus
              OR Avt_SHU_vkl.topStatus
              OR All_IM_Off.topStatus
              OR Nalichie220_SHU_Ai.topStatus
              OR BP_Norm.topStatus
              OR Naprajenie_U_IM.topStatus
              OR MV_Poloj_RolledON.topStatus
              OR MV_Poloj_RolledOFF.topStatus
              OR NOTAnalogNS.topStatus
              OR Net_ASPS_Analogs.topStatus
              OR Not_AS.topStatus
              OR Gotov_Vozb.topStatus
              OR Reactornyi_P.topStatus
              OR Chastotnyi_P.topStatus
              OR dP_kr1.topStatus
              OR Auto_Rej.topStatus
              OR CK_IM_Norm.topStatus
              OR HAnd_Mode.topStatus
              OR Impuls_Gaz.topStatus;

  (*TODO: TYPE PROGRAM CODE HERE*)
  StrAlg.status :=  SHL(BYTE_TO_DWORD(source_for_Status), 29)
  			OR SHL(BYTE_TO_DWORD(cmd_for_Status), 26)
  			OR SHL(BYTE_TO_DWORD(command_error_for_Status), 23)
  			OR SHL(BOOL_TO_DWORD(StrAlg.OpcCommandsDisabled ), 21)
                                OR SHL(BOOL_TO_DWORD(testAllowed),16)
                                OR SHL(BOOL_TO_DWORD(puskAllowed),15)
  			OR SHL(BOOL_TO_DWORD(StrAlg.hasError),4)
  			OR SHL(BOOL_TO_DWORD(StrAlg.CanRun),2)
  			OR SHL(BOOL_TO_DWORD(StrAlg.isEnded),1)
  			OR BOOL_TO_DWORD(StrAlg.isRuning);
END_FUNCTION_BLOCK

FUNCTION_BLOCK fillingAlg
  VAR_IN_OUT
    StrAlg : struct_Alg;
  END_VAR
  VAR
    BreakPuskTimer : struct_PhaseAlgoritm;
    kran3bOpen : struct_PhaseAlgoritm;
    kran4Open : struct_PhaseAlgoritm;
    waitAfterKran4 : struct_PhaseAlgoritm;
    kran5Close : struct_PhaseAlgoritm;
    didPKran1 : struct_PhaseAlgoritm;
    kran1Open : struct_PhaseAlgoritm;
    kran2Open : struct_PhaseAlgoritm;
    kran3bClose : struct_PhaseAlgoritm;
    kran4Close : struct_PhaseAlgoritm;
    RunProtection_kr1 : struct_PhaseAlgoritm;
    RunProtection_kr2 : struct_PhaseAlgoritm;
    waitAfterKran5 : struct_PhaseAlgoritm;
    testUnsuccessfulFilling : struct_PhaseAlgoritm;
    fb_BreakPuskTimer : fb_ph_Timer;
    fb_kran3bOpen : fb_ph_Kran;
    fb_kran4Open : fb_ph_Kran;
    fb_waitAfterKran4 : fb_ph_Timer;
    fb_kran5Close : fb_ph_Kran;
    fb_didPKran1 : fb_ph_CustomPhase;
    fb_kran1Open : fb_ph_Kran;
    fb_kran2Open : fb_ph_Kran;
    fb_kran3bClose : fb_ph_Kran;
    fb_kran4Close : fb_ph_Kran;
    fb_RunProtection_kr1 : fb_ph_DIprotection;
    fb_RunProtection_kr2 : fb_ph_DIprotection;
    fb_waitAfterKran5 : fb_ph_Timer;
    fb_testUnsuccessfulFilling : fb_ph_CustomPhase;
    _sunpackerCommand : fb_sunpackerCommand;
    _DualStateImAction : TYPE_DualStateImAction;
    _PhaseAlgoritmAction : TYPE_PhaseAlgoritmAction;
    source : BYTE;
    cmd : BYTE;
    lastCmd : BYTE;
    source_for_Status : BYTE;
    cmd_for_Status : BYTE;
    command_error_for_Status : BYTE;
    resetCmdTimer : TON;
    resetCmdTimerPriznak : BOOL;
    onInit : BOOL;
    waitReset : TON;
  END_VAR
  VAR_EXTERNAL
    IM : ImConfig;
    ai : AiConfig;
    protections : ProtectionsConfig;
    AlgTimers : struct_AlgTimers;
    algoritms : AlgoritmsConfig;
  END_VAR

  IF NOT onInit THEN

           fb_BreakPuskTimer(phaseNumber:=0, delay:=T#240S);
               fb_kran3bOpen(phaseNumber:=1, act:=_on);
                fb_kran4Open(phaseNumber:=2, act:=_on);
           fb_waitAfterKran4(phaseNumber:=3, delay:=T#10S);
               fb_kran5Close(phaseNumber:=4, act:=_off);
                fb_didPKran1(phaseNumber:=5);
                fb_kran1Open(phaseNumber:=7, act:=_on);
                fb_kran2Open(phaseNumber:=8, act:=_on);
              fb_kran3bClose(phaseNumber:=9, act:=_off);
               fb_kran4Close(phaseNumber:=10, act:=_off);
        fb_RunProtection_kr1(phaseNumber:=11, act:=_run);
        fb_RunProtection_kr2(phaseNumber:=12, act:=_run);
           fb_waitAfterKran5(phaseNumber:=13, delay:=T#60S);
  fb_testUnsuccessfulFilling(phaseNumber:=17);

  onInit:=TRUE;
  END_IF;

           fb_BreakPuskTimer(StrPh:=BreakPuskTimer, timer:=AlgTimers.filling_BreakPuskTimer);
               fb_kran3bOpen(StrPh:=kran3bOpen, Im:=Im.kran3b);
                fb_kran4Open(StrPh:=kran4Open, Im:=Im.kran4);
           fb_waitAfterKran4(StrPh:=waitAfterKran4, timer:=AlgTimers.filling_waitAfterKran4);
               fb_kran5Close(StrPh:=kran5Close, Im:=Im.kran5);
                fb_didPKran1(StrPh:=didPKran1);
                fb_kran1Open(StrPh:=kran1Open, Im:=Im.kran1);
                fb_kran2Open(StrPh:=kran2Open, Im:=Im.kran2);
              fb_kran3bClose(StrPh:=kran3bClose, Im:=Im.kran3b);
               fb_kran4Close(StrPh:=kran4Close, Im:=Im.kran4);
        fb_RunProtection_kr1(StrPh:=RunProtection_kr1 , StrDiP:=protections.Reg_vozb_off);
        fb_RunProtection_kr2(StrPh:=RunProtection_kr2 , StrDiP:=protections.Fail_chastotnii_pusk);
           fb_waitAfterKran5(StrPh:=waitAfterKran5, timer:=AlgTimers.filling_waitAfterKran5);
  fb_testUnsuccessfulFilling(StrPh:=testUnsuccessfulFilling);
